LIN {X 0,Y 488.673,Z 877.462,A -85,B 0,C 180,E1 10645.22,E2 10645.22} C_VEL
LIN {X 0,Y 505.067,Z 659.216,A -85,B 0,C 180,E1 10641.829,E2 10641.829} C_VEL
LIN {X 0,Y 508.295,Z 617.041,A -85,B 0,C 180,E1 10641.16,E2 10641.16} C_VEL
LIN {X 0,Y 501.878,Z 605.856,A -85,B 0,C 180,E1 10638.709,E2 10638.709} C_VEL
LIN {X 0,Y 495.396,Z 596.132,A -85,B 0,C 180,E1 10635.872,E2 10635.872} C_VEL
LIN {X 0,Y 491.953,Z 591.127,A -85,B 0,C 180,E1 10634.117,E2 10634.117} C_VEL
LIN {X 0,Y 489.104,Z 586.88,A -85,B 0,C 180,E1 10632.455,E2 10632.455} C_VEL
LIN {X 0,Y 486.126,Z 582.532,A -85,B 0,C 180,E1 10630.428,E2 10630.428} C_VEL
LIN {X 0,Y 483.244,Z 578.317,A -85,B 0,C 180,E1 10627.969,E2 10627.969} C_VEL
LIN {X 0,Y 482.559,Z 577.333,A -85,B 0,C 180,E1 10627.261,E2 10627.261} C_VEL
LIN {X 0,Y 479.956,Z 573.698,A -85,B 0,C 180,E1 10623.464,E2 10623.464} C_VEL
LIN {X 0,Y 479.541,Z 571.93,A -85,B 0,C 180,E1 10621.912,E2 10621.912} C_VEL
LIN {X 0,Y 479.637,Z 572.192,A -85,B 0,C 180,E1 10617.491,E2 10617.491} C_VEL
LIN {X 0,Y 481.251,Z 576.101,A -85,B 0,C 180,E1 10614.037,E2 10614.037} C_VEL
LIN {X 0,Y 483.062,Z 577.924,A -85,B 0,C 180,E1 10612.028,E2 10612.028} C_VEL
LIN {X 0,Y 485.863,Z 582.227,A -85,B 0,C 180,E1 10609.566,E2 10609.566} C_VEL
LIN {X 0,Y 486.983,Z 583.755,A -85,B 0,C 180,E1 10608.752,E2 10608.752} C_VEL
LIN {X 0,Y 490.511,Z 588.903,A -85,B 0,C 180,E1 10606.502,E2 10606.502} C_VEL
LIN {X 0,Y 494.214,Z 594.346,A -85,B 0,C 180,E1 10604.51,E2 10604.51} C_VEL
LIN {X 0,Y 499.508,Z 602.191,A -85,B 0,C 180,E1 10602.075,E2 10602.075} C_VEL
LIN {X 0,Y 505.798,Z 612.068,A -85,B 0,C 180,E1 10599.579,E2 10599.579} C_VEL
LIN {X 0,Y 508.298,Z 616.319,A -85,B 0,C 180,E1 10598.668,E2 10598.668} C_VEL
LIN {X 0,Y 491.94,Z 831.282,A -85,B 0,C 180,E1 10595.331,E2 10595.331} C_VEL
LIN {X 0,Y 486.711,Z 898.786,A -85,B 0,C 180,E1 10594.263,E2 10594.263} C_VEL
LIN {X 0,Y 482.885,Z 928.156,A -85,B 0,C 180,E1 10593.691,E2 10593.691} C_VEL
LIN {X 0,Y 478.634,Z 951.918,A -85,B 0,C 180,E1 10593.081,E2 10593.081} C_VEL
LIN {X 0,Y 474.12,Z 972.963,A -85,B 0,C 180,E1 10592.412,E2 10592.412} C_VEL
LIN {X 0,Y 468.985,Z 993.591,A -85,B 0,C 180,E1 10591.626,E2 10591.626} C_VEL
LIN {X 0,Y 461.912,Z 1018.559,A -85,B 0,C 180,E1 10590.484,E2 10590.484} C_VEL
LIN {X 0,Y 453.841,Z 1042.99,A -85,B 0,C 180,E1 10589.113,E2 10589.113} C_VEL
LIN {X 0,Y 446.612,Z 1062.769,A -85,B 0,C 180,E1 10587.812,E2 10587.812} C_VEL
LIN {X 0,Y 439.339,Z 1081.192,A -85,B 0,C 180,E1 10586.408,E2 10586.408} C_VEL
LIN {X 0,Y 431.297,Z 1100.199,A -85,B 0,C 180,E1 10584.741,E2 10584.741} C_VEL
LIN {X 0,Y 420.775,Z 1123.256,A -85,B 0,C 180,E1 10582.359,E2 10582.359} C_VEL
LIN {X 0,Y 412.35,Z 1140.615,A -85,B 0,C 180,E1 10580.238,E2 10580.238} C_VEL
LIN {X 0,Y 404.56,Z 1156.078,A -85,B 0,C 180,E1 10578.071,E2 10578.071} C_VEL
LIN {X 0,Y 396.87,Z 1170.932,A -85,B 0,C 180,E1 10575.689,E2 10575.689} C_VEL
LIN {X 0,Y 387.854,Z 1188.135,A -85,B 0,C 180,E1 10572.491,E2 10572.491} C_VEL
LIN {X 0,Y 379.872,Z 1203.044,A -85,B 0,C 180,E1 10569.181,E2 10569.181} C_VEL
LIN {X 0,Y 373.901,Z 1214.52,A -85,B 0,C 180,E1 10566.231,E2 10566.231} C_VEL
LIN {X 0,Y 368.717,Z 1224.76,A -85,B 0,C 180,E1 10563.219,E2 10563.219} C_VEL
LIN {X 0,Y 363.893,Z 1234.761,A -85,B 0,C 180,E1 10559.828,E2 10559.828} C_VEL
LIN {X 0,Y 359.105,Z 1245.725,A -85,B 0,C 180,E1 10555.395,E2 10555.395} C_VEL
LIN {X 0,Y 356.135,Z 1253.418,A -85,B 0,C 180,E1 10551.584,E2 10551.584} C_VEL
LIN {X 0,Y 354.269,Z 1259.29,A -85,B 0,C 180,E1 10548.091,E2 10548.091} C_VEL
LIN {X 0,Y 353.032,Z 1264.082,A -85,B 0,C 180,E1 10544.604,E2 10544.604} C_VEL
LIN {X 0,Y 352.351,Z 1267.827,A -85,B 0,C 180,E1 10541.13,E2 10541.13} C_VEL
LIN {X 0,Y 352.013,Z 1270.668,A -85,B 0,C 180,E1 10537.512,E2 10537.512} C_VEL
LIN {X 0,Y 351.926,Z 1272.49,A -85,B 0,C 180,E1 10533.751,E2 10533.751} C_VEL
LIN {X 0,Y 351.896,Z 1273.142,A -85,B 0,C 180,E1 10529.842,E2 10529.842} C_VEL
LIN {X 0,Y 351.929,Z 1272.4,A -85,B 0,C 180,E1 10525.932,E2 10525.932} C_VEL
LIN {X 0,Y 352.019,Z 1270.629,A -85,B 0,C 180,E1 10522.333,E2 10522.333} C_VEL
LIN {X 0,Y 352.334,Z 1267.928,A -85,B 0,C 180,E1 10518.879,E2 10518.879} C_VEL
LIN {X 0,Y 353.012,Z 1264.211,A -85,B 0,C 180,E1 10515.404,E2 10515.404} C_VEL
LIN {X 0,Y 354.153,Z 1259.69,A -85,B 0,C 180,E1 10512.076,E2 10512.076} C_VEL
LIN {X 0,Y 355.968,Z 1253.906,A -85,B 0,C 180,E1 10508.589,E2 10508.589} C_VEL
LIN {X 0,Y 358.586,Z 1246.992,A -85,B 0,C 180,E1 10505.105,E2 10505.105} C_VEL
LIN {X 0,Y 361.326,Z 1240.495,A -85,B 0,C 180,E1 10502.297,E2 10502.297} C_VEL
LIN {X 0,Y 361.626,Z 1237.874,A -85,B 0,C 180,E1 10501.14,E2 10501.14} C_VEL
LIN {X 0,Y 359.431,Z 1230.835,A -85,B 0,C 180,E1 10497.968,E2 10497.968} C_VEL
LIN {X 0,Y 360.102,Z 1228.131,A -85,B 0,C 180,E1 10497.004,E2 10497.004} C_VEL
LIN {X 0,Y 366.407,Z 1216.08,A -85,B 0,C 180,E1 10493.307,E2 10493.307} C_VEL
LIN {X 0,Y 372.543,Z 1204.763,A -85,B 0,C 180,E1 10490.307,E2 10490.307} C_VEL
LIN {X 0,Y 379.15,Z 1192.807,A -85,B 0,C 180,E1 10487.545,E2 10487.545} C_VEL
LIN {X 0,Y 387.197,Z 1178.247,A -85,B 0,C 180,E1 10484.621,E2 10484.621} C_VEL
LIN {X 0,Y 397.614,Z 1158.992,A -85,B 0,C 180,E1 10481.363,E2 10481.363} C_VEL
LIN {X 0,Y 406.081,Z 1142.782,A -85,B 0,C 180,E1 10479.037,E2 10479.037} C_VEL
LIN {X 0,Y 414.037,Z 1126.962,A -85,B 0,C 180,E1 10477.057,E2 10477.057} C_VEL
LIN {X 0,Y 422.44,Z 1109.459,A -85,B 0,C 180,E1 10475.148,E2 10475.148} C_VEL
LIN {X 0,Y 432.786,Z 1086.479,A -85,B 0,C 180,E1 10473.013,E2 10473.013} C_VEL
LIN {X 0,Y 441.432,Z 1065.351,A -85,B 0,C 180,E1 10471.369,E2 10471.369} C_VEL
LIN {X 0,Y 448.646,Z 1046.297,A -85,B 0,C 180,E1 10470.096,E2 10470.096} C_VEL
LIN {X 0,Y 455.36,Z 1026.795,A -85,B 0,C 180,E1 10468.963,E2 10468.963} C_VEL
LIN {X 0,Y 462.1,Z 1005.168,A -85,B 0,C 180,E1 10467.895,E2 10467.895} C_VEL
LIN {X 0,Y 469.494,Z 977.542,A -85,B 0,C 180,E1 10466.775,E2 10466.775} C_VEL
LIN {X 0,Y 474.536,Z 955.094,A -85,B 0,C 180,E1 10466.047,E2 10466.047} C_VEL
LIN {X 0,Y 478.563,Z 933.64,A -85,B 0,C 180,E1 10465.477,E2 10465.477} C_VEL
LIN {X 0,Y 481.975,Z 911.074,A -85,B 0,C 180,E1 10465.003,E2 10465.003} C_VEL
LIN {X 0,Y 485.059,Z 880.548,A -85,B 0,C 180,E1 10464.481,E2 10464.481} C_VEL
LIN {X 0,Y 502.082,Z 660.192,A -85,B 0,C 180,E1 10461.066,E2 10461.066} C_VEL
LIN {X 0,Y 505.159,Z 621.258,A -85,B 0,C 180,E1 10460.454,E2 10460.454} C_VEL
LIN {X 0,Y 498.577,Z 610.88,A -85,B 0,C 180,E1 10457.839,E2 10457.839} C_VEL
LIN {X 0,Y 493.32,Z 602.856,A -85,B 0,C 180,E1 10455.398,E2 10455.398} C_VEL
LIN {X 0,Y 490.433,Z 598.562,A -85,B 0,C 180,E1 10453.861,E2 10453.861} C_VEL
LIN {X 0,Y 487.858,Z 594.642,A -85,B 0,C 180,E1 10452.307,E2 10452.307} C_VEL
LIN {X 0,Y 485.045,Z 590.425,A -85,B 0,C 180,E1 10450.332,E2 10450.332} C_VEL
LIN {X 0,Y 482.19,Z 586.179,A -85,B 0,C 180,E1 10447.806,E2 10447.806} C_VEL
LIN {X 0,Y 481.587,Z 585.291,A -85,B 0,C 180,E1 10447.156,E2 10447.156} C_VEL
LIN {X 0,Y 479.07,Z 581.699,A -85,B 0,C 180,E1 10443.231,E2 10443.231} C_VEL
LIN {X 0,Y 478.717,Z 579.913,A -85,B 0,C 180,E1 10441.556,E2 10441.556} C_VEL
LIN {X 0,Y 478.774,Z 580.143,A -85,B 0,C 180,E1 10438.205,E2 10438.205} C_VEL
LIN {X 0,Y 480.295,Z 584.064,A -85,B 0,C 180,E1 10434.505,E2 10434.505} C_VEL
LIN {X 0,Y 482.075,Z 585.927,A -85,B 0,C 180,E1 10432.432,E2 10432.432} C_VEL
LIN {X 0,Y 484.713,Z 590.12,A -85,B 0,C 180,E1 10430.021,E2 10430.021} C_VEL
LIN {X 0,Y 485.887,Z 591.683,A -85,B 0,C 180,E1 10429.147,E2 10429.147} C_VEL
LIN {X 0,Y 489.137,Z 596.588,A -85,B 0,C 180,E1 10427.005,E2 10427.005} C_VEL
LIN {X 0,Y 492.963,Z 602.326,A -85,B 0,C 180,E1 10424.892,E2 10424.892} C_VEL
LIN {X 0,Y 497.914,Z 609.822,A -85,B 0,C 180,E1 10422.559,E2 10422.559} C_VEL
LIN {X 0,Y 502.016,Z 616.506,A -85,B 0,C 180,E1 10420.844,E2 10420.844} C_VEL
LIN {X 0,Y 505.192,Z 622.48,A -85,B 0,C 180,E1 10419.596,E2 10419.596} C_VEL
LIN {X 0,Y 488.383,Z 838.103,A -85,B 0,C 180,E1 10416.255,E2 10416.255} C_VEL
LIN {X 0,Y 483.187,Z 903.482,A -85,B 0,C 180,E1 10415.22,E2 10415.22} C_VEL
LIN {X 0,Y 479.179,Z 933.314,A -85,B 0,C 180,E1 10414.646,E2 10414.646} C_VEL
LIN {X 0,Y 474.882,Z 956.587,A -85,B 0,C 180,E1 10414.066,E2 10414.066} C_VEL
LIN {X 0,Y 470.159,Z 977.971,A -85,B 0,C 180,E1 10413.403,E2 10413.403} C_VEL
LIN {X 0,Y 464.921,Z 998.45,A -85,B 0,C 180,E1 10412.638,E2 10412.638} C_VEL
LIN {X 0,Y 458.057,Z 1022.054,A -85,B 0,C 180,E1 10411.584,E2 10411.584} C_VEL
LIN {X 0,Y 449.414,Z 1047.74,A -85,B 0,C 180,E1 10410.18,E2 10410.18} C_VEL
LIN {X 0,Y 441.99,Z 1067.639,A -85,B 0,C 180,E1 10408.887,E2 10408.887} C_VEL
LIN {X 0,Y 434.502,Z 1086.202,A -85,B 0,C 180,E1 10407.489,E2 10407.489} C_VEL
LIN {X 0,Y 426.73,Z 1104.125,A -85,B 0,C 180,E1 10405.943,E2 10405.943} C_VEL
LIN {X 0,Y 416.615,Z 1126.069,A -85,B 0,C 180,E1 10403.736,E2 10403.736} C_VEL
LIN {X 0,Y 406.825,Z 1145.735,A -85,B 0,C 180,E1 10401.37,E2 10401.37} C_VEL
LIN {X 0,Y 398.797,Z 1161.288,A -85,B 0,C 180,E1 10399.208,E2 10399.208} C_VEL
LIN {X 0,Y 390.814,Z 1176.347,A -85,B 0,C 180,E1 10396.807,E2 10396.807} C_VEL
LIN {X 0,Y 381.815,Z 1193.118,A -85,B 0,C 180,E1 10393.715,E2 10393.715} C_VEL
LIN {X 0,Y 373.067,Z 1209.073,A -85,B 0,C 180,E1 10390.195,E2 10390.195} C_VEL
LIN {X 0,Y 366.564,Z 1221.218,A -85,B 0,C 180,E1 10387.065,E2 10387.065} C_VEL
LIN {X 0,Y 360.942,Z 1232.107,A -85,B 0,C 180,E1 10383.828,E2 10383.828} C_VEL
LIN {X 0,Y 355.178,Z 1244.038,A -85,B 0,C 180,E1 10379.694,E2 10379.694} C_VEL
LIN {X 0,Y 350.781,Z 1253.927,A -85,B 0,C 180,E1 10375.488,E2 10375.488} C_VEL
LIN {X 0,Y 348.032,Z 1261.068,A -85,B 0,C 180,E1 10371.878,E2 10371.878} C_VEL
LIN {X 0,Y 346.177,Z 1266.915,A -85,B 0,C 180,E1 10368.345,E2 10368.345} C_VEL
LIN {X 0,Y 344.975,Z 1271.541,A -85,B 0,C 180,E1 10364.943,E2 10364.943} C_VEL
LIN {X 0,Y 344.322,Z 1275.199,A -85,B 0,C 180,E1 10361.553,E2 10361.553} C_VEL
LIN {X 0,Y 343.989,Z 1278.028,A -85,B 0,C 180,E1 10358.015,E2 10358.015} C_VEL
LIN {X 0,Y 343.923,Z 1279.699,A -85,B 0,C 180,E1 10354.831,E2 10354.831} C_VEL
LIN {X 0,Y 343.908,Z 1280.543,A -85,B 0,C 180,E1 10351.661,E2 10351.661} C_VEL
LIN {X 0,Y 343.905,Z 1280.564,A -85,B 0,C 180,E1 10348.496,E2 10348.496} C_VEL
LIN {X 0,Y 343.921,Z 1279.761,A -85,B 0,C 180,E1 10345.326,E2 10345.326} C_VEL
LIN {X 0,Y 343.984,Z 1278.131,A -85,B 0,C 180,E1 10342.143,E2 10342.143} C_VEL
LIN {X 0,Y 344.302,Z 1275.345,A -85,B 0,C 180,E1 10338.606,E2 10338.606} C_VEL
LIN {X 0,Y 344.94,Z 1271.729,A -85,B 0,C 180,E1 10335.217,E2 10335.217} C_VEL
LIN {X 0,Y 346.108,Z 1267.147,A -85,B 0,C 180,E1 10331.816,E2 10331.816} C_VEL
LIN {X 0,Y 347.852,Z 1261.567,A -85,B 0,C 180,E1 10328.408,E2 10328.408} C_VEL
LIN {X 0,Y 350.353,Z 1254.956,A -85,B 0,C 180,E1 10325.011,E2 10325.011} C_VEL
LIN {X 0,Y 353.834,Z 1246.86,A -85,B 0,C 180,E1 10321.469,E2 10321.469} C_VEL
LIN {X 0,Y 359.203,Z 1235.669,A -85,B 0,C 180,E1 10317.311,E2 10317.311} C_VEL
LIN {X 0,Y 365.688,Z 1222.885,A -85,B 0,C 180,E1 10313.407,E2 10313.407} C_VEL
LIN {X 0,Y 372.086,Z 1210.809,A -85,B 0,C 180,E1 10310.237,E2 10310.237} C_VEL
LIN {X 0,Y 379.059,Z 1197.97,A -85,B 0,C 180,E1 10307.315,E2 10307.315} C_VEL
LIN {X 0,Y 388.176,Z 1181.321,A -85,B 0,C 180,E1 10304.052,E2 10304.052} C_VEL
LIN {X 0,Y 397.622,Z 1163.448,A -85,B 0,C 180,E1 10301.126,E2 10301.126} C_VEL
LIN {X 0,Y 405.541,Z 1148.136,A -85,B 0,C 180,E1 10298.956,E2 10298.956} C_VEL
LIN {X 0,Y 413.295,Z 1132.58,A -85,B 0,C 180,E1 10297.022,E2 10297.022} C_VEL
LIN {X 0,Y 421.7,Z 1114.95,A -85,B 0,C 180,E1 10295.109,E2 10295.109} C_VEL
LIN {X 0,Y 431.768,Z 1092.578,A -85,B 0,C 180,E1 10293.034,E2 10293.034} C_VEL
LIN {X 0,Y 440.736,Z 1070.608,A -85,B 0,C 180,E1 10291.33,E2 10291.33} C_VEL
LIN {X 0,Y 448.129,Z 1051.038,A -85,B 0,C 180,E1 10290.032,E2 10290.032} C_VEL
LIN {X 0,Y 454.755,Z 1031.833,A -85,B 0,C 180,E1 10288.929,E2 10288.929} C_VEL
LIN {X 0,Y 461.501,Z 1010.238,A -85,B 0,C 180,E1 10287.872,E2 10287.872} C_VEL
LIN {X 0,Y 468.956,Z 982.613,A -85,B 0,C 180,E1 10286.765,E2 10286.765} C_VEL
LIN {X 0,Y 474.149,Z 959.6,A -85,B 0,C 180,E1 10286.027,E2 10286.027} C_VEL
LIN {X 0,Y 478.201,Z 938.258,A -85,B 0,C 180,E1 10285.474,E2 10285.474} C_VEL
LIN {X 0,Y 481.638,Z 915.668,A -85,B 0,C 180,E1 10285.006,E2 10285.006} C_VEL
LIN {X 0,Y 484.693,Z 885.505,A -85,B 0,C 180,E1 10284.489,E2 10284.489} C_VEL
LIN {X 0,Y 501.542,Z 666.545,A -85,B 0,C 180,E1 10281.092,E2 10281.092} C_VEL
LIN {X 0,Y 505.043,Z 622.093,A -85,B 0,C 180,E1 10280.392,E2 10280.392} C_VEL
LIN {X 0,Y 499.654,Z 612.643,A -85,B 0,C 180,E1 10278.251,E2 10278.251} C_VEL
LIN {X 0,Y 493.706,Z 603.514,A -85,B 0,C 180,E1 10275.566,E2 10275.566} C_VEL
LIN {X 0,Y 490.446,Z 598.675,A -85,B 0,C 180,E1 10273.86,E2 10273.86} C_VEL
LIN {X 0,Y 487.658,Z 594.454,A -85,B 0,C 180,E1 10272.192,E2 10272.192} C_VEL
LIN {X 0,Y 484.832,Z 590.256,A -85,B 0,C 180,E1 10270.216,E2 10270.216} C_VEL
LIN {X 0,Y 482.032,Z 586.005,A -85,B 0,C 180,E1 10267.749,E2 10267.749} C_VEL
LIN {X 0,Y 481.027,Z 584.85,A -85,B 0,C 180,E1 10266.685,E2 10266.685} C_VEL
LIN {X 0,Y 478.85,Z 581.273,A -85,B 0,C 180,E1 10263.112,E2 10263.112} C_VEL
LIN {X 0,Y 478.533,Z 579.863,A -85,B 0,C 180,E1 10261.796,E2 10261.796} C_VEL
LIN {X 0,Y 478.629,Z 580.078,A -85,B 0,C 180,E1 10257.605,E2 10257.605} C_VEL
LIN {X 0,Y 480.188,Z 583.98,A -85,B 0,C 180,E1 10254.144,E2 10254.144} C_VEL
LIN {X 0,Y 481.908,Z 585.739,A -85,B 0,C 180,E1 10252.189,E2 10252.189} C_VEL
LIN {X 0,Y 484.732,Z 590.11,A -85,B 0,C 180,E1 10249.662,E2 10249.662} C_VEL
LIN {X 0,Y 486.15,Z 592.291,A -85,B 0,C 180,E1 10248.612,E2 10248.612} C_VEL
LIN {X 0,Y 489.131,Z 596.606,A -85,B 0,C 180,E1 10246.704,E2 10246.704} C_VEL
LIN {X 0,Y 492.773,Z 602.066,A -85,B 0,C 180,E1 10244.705,E2 10244.705} C_VEL
LIN {X 0,Y 497.925,Z 609.877,A -85,B 0,C 180,E1 10242.288,E2 10242.288} C_VEL
LIN {X 0,Y 504.13,Z 619.794,A -85,B 0,C 180,E1 10239.781,E2 10239.781} C_VEL
LIN {X 0,Y 505.034,Z 621.396,A -85,B 0,C 180,E1 10239.439,E2 10239.439} C_VEL
LIN {X 0,Y 488.271,Z 836.362,A -85,B 0,C 180,E1 10236.108,E2 10236.108} C_VEL
LIN {X 0,Y 483.251,Z 899.218,A -85,B 0,C 180,E1 10235.114,E2 10235.114} C_VEL
LIN {X 0,Y 479.184,Z 929.39,A -85,B 0,C 180,E1 10234.525,E2 10234.525} C_VEL
LIN {X 0,Y 474.979,Z 952.343,A -85,B 0,C 180,E1 10233.937,E2 10233.937} C_VEL
LIN {X 0,Y 470.439,Z 973.061,A -85,B 0,C 180,E1 10233.282,E2 10233.282} C_VEL
LIN {X 0,Y 465.241,Z 993.523,A -85,B 0,C 180,E1 10232.509,E2 10232.509} C_VEL
LIN {X 0,Y 458.3,Z 1017.528,A -85,B 0,C 180,E1 10231.422,E2 10231.422} C_VEL
LIN {X 0,Y 450.024,Z 1042.211,A -85,B 0,C 180,E1 10230.06,E2 10230.06} C_VEL
LIN {X 0,Y 442.625,Z 1062.056,A -85,B 0,C 180,E1 10228.766,E2 10228.766} C_VEL
LIN {X 0,Y 435.084,Z 1080.742,A -85,B 0,C 180,E1 10227.352,E2 10227.352} C_VEL
LIN {X 0,Y 427.356,Z 1098.571,A -85,B 0,C 180,E1 10225.804,E2 10225.804} C_VEL
LIN {X 0,Y 417.616,Z 1119.697,A -85,B 0,C 180,E1 10223.678,E2 10223.678} C_VEL
LIN {X 0,Y 407.616,Z 1139.7,A -85,B 0,C 180,E1 10221.269,E2 10221.269} C_VEL
LIN {X 0,Y 399.533,Z 1155.251,A -85,B 0,C 180,E1 10219.098,E2 10219.098} C_VEL
LIN {X 0,Y 391.985,Z 1169.345,A -85,B 0,C 180,E1 10216.851,E2 10216.851} C_VEL
LIN {X 0,Y 384.158,Z 1183.682,A -85,B 0,C 180,E1 10214.234,E2 10214.234} C_VEL
LIN {X 0,Y 375.224,Z 1199.984,A -85,B 0,C 180,E1 10210.762,E2 10210.762} C_VEL
LIN {X 0,Y 367.775,Z 1213.475,A -85,B 0,C 180,E1 10207.325,E2 10207.325} C_VEL
LIN {X 0,Y 361.994,Z 1224.343,A -85,B 0,C 180,E1 10204.109,E2 10204.109} C_VEL
LIN {X 0,Y 357.11,Z 1233.945,A -85,B 0,C 180,E1 10200.827,E2 10200.827} C_VEL
LIN {X 0,Y 352.434,Z 1243.967,A -85,B 0,C 180,E1 10196.818,E2 10196.818} C_VEL
LIN {X 0,Y 348.697,Z 1252.91,A -85,B 0,C 180,E1 10192.423,E2 10192.423} C_VEL
LIN {X 0,Y 346.534,Z 1259.129,A -85,B 0,C 180,E1 10188.684,E2 10188.684} C_VEL
LIN {X 0,Y 345.213,Z 1263.764,A -85,B 0,C 180,E1 10185.287,E2 10185.287} C_VEL
LIN {X 0,Y 344.465,Z 1267.443,A -85,B 0,C 180,E1 10181.898,E2 10181.898} C_VEL
LIN {X 0,Y 344.056,Z 1270.308,A -85,B 0,C 180,E1 10178.36,E2 10178.36} C_VEL
LIN {X 0,Y 343.944,Z 1272.041,A -85,B 0,C 180,E1 10175.175,E2 10175.175} C_VEL
LIN {X 0,Y 343.913,Z 1272.968,A -85,B 0,C 180,E1 10172.004,E2 10172.004} C_VEL
LIN {X 0,Y 343.888,Z 1273.095,A -85,B 0,C 180,E1 10168.839,E2 10168.839} C_VEL
LIN {X 0,Y 343.932,Z 1272.353,A -85,B 0,C 180,E1 10165.503,E2 10165.503} C_VEL
LIN {X 0,Y 344.023,Z 1270.717,A -85,B 0,C 180,E1 10162.154,E2 10162.154} C_VEL
LIN {X 0,Y 344.373,Z 1268.017,A -85,B 0,C 180,E1 10158.618,E2 10158.618} C_VEL
LIN {X 0,Y 345.058,Z 1264.504,A -85,B 0,C 180,E1 10155.232,E2 10155.232} C_VEL
LIN {X 0,Y 346.269,Z 1260.005,A -85,B 0,C 180,E1 10151.81,E2 10151.81} C_VEL
LIN {X 0,Y 348.165,Z 1254.296,A -85,B 0,C 180,E1 10148.261,E2 10148.261} C_VEL
LIN {X 0,Y 350.757,Z 1247.782,A -85,B 0,C 180,E1 10144.872,E2 10144.872} C_VEL
LIN {X 0,Y 354.526,Z 1239.394,A -85,B 0,C 180,E1 10141.172,E2 10141.172} C_VEL
LIN {X 0,Y 360.102,Z 1228.131,A -85,B 0,C 180,E1 10137.004,E2 10137.004} C_VEL
LIN {X 0,Y 360.852,Z 1224.964,A -85,B 0,C 180,E1 10135.886,E2 10135.886} C_VEL
LIN {X 0,Y 359.897,Z 1217.295,A -85,B 0,C 180,E1 10132.928,E2 10132.928} C_VEL
LIN {X 0,Y 361.031,Z 1213.805,A -85,B 0,C 180,E1 10131.835,E2 10131.835} C_VEL
LIN {X 0,Y 369.435,Z 1199.299,A -85,B 0,C 180,E1 10128.099,E2 10128.099} C_VEL
LIN {X 0,Y 378.439,Z 1183.444,A -85,B 0,C 180,E1 10124.714,E2 10124.714} C_VEL
LIN {X 0,Y 386.113,Z 1169.91,A -85,B 0,C 180,E1 10122.224,E2 10122.224} C_VEL
LIN {X 0,Y 393.936,Z 1155.806,A -85,B 0,C 180,E1 10119.954,E2 10119.954} C_VEL
LIN {X 0,Y 402.042,Z 1140.729,A -85,B 0,C 180,E1 10117.831,E2 10117.831} C_VEL
LIN {X 0,Y 411.334,Z 1122.726,A -85,B 0,C 180,E1 10115.631,E2 10115.631} C_VEL
LIN {X 0,Y 422.245,Z 1100.052,A -85,B 0,C 180,E1 10113.3,E2 10113.3} C_VEL
LIN {X 0,Y 430.24,Z 1082.169,A -85,B 0,C 180,E1 10111.736,E2 10111.736} C_VEL
LIN {X 0,Y 437.872,Z 1063.817,A -85,B 0,C 180,E1 10110.338,E2 10110.338} C_VEL
LIN {X 0,Y 445.433,Z 1044.138,A -85,B 0,C 180,E1 10109.047,E2 10109.047} C_VEL
LIN {X 0,Y 453.195,Z 1021.864,A -85,B 0,C 180,E1 10107.795,E2 10107.795} C_VEL
LIN {X 0,Y 461.151,Z 995.561,A -85,B 0,C 180,E1 10106.582,E2 10106.582} C_VEL
LIN {X 0,Y 466.66,Z 974.518,A -85,B 0,C 180,E1 10105.783,E2 10105.783} C_VEL
LIN {X 0,Y 471.412,Z 953.438,A -85,B 0,C 180,E1 10105.116,E2 10105.116} C_VEL
LIN {X 0,Y 475.529,Z 931.632,A -85,B 0,C 180,E1 10104.554,E2 10104.554} C_VEL
LIN {X 0,Y 479.571,Z 904.31,A -85,B 0,C 180,E1 10104.003,E2 10104.003} C_VEL
LIN {X 0,Y 483.419,Z 859.466,A -85,B 0,C 180,E1 10103.284,E2 10103.284} C_VEL
LIN {X 0,Y 500.832,Z 640.859,A -85,B 0,C 180,E1 10099.906,E2 10099.906} C_VEL
LIN {X 0,Y 501.967,Z 626.544,A -85,B 0,C 180,E1 10099.672,E2 10099.672} C_VEL
LIN {X 0,Y 495.879,Z 616.663,A -85,B 0,C 180,E1 10097.121,E2 10097.121} C_VEL
LIN {X 0,Y 489.971,Z 607.504,A -85,B 0,C 180,E1 10094.175,E2 10094.175} C_VEL
LIN {X 0,Y 486.334,Z 602.099,A -85,B 0,C 180,E1 10091.985,E2 10091.985} C_VEL
LIN {X 0,Y 483.758,Z 598.151,A -85,B 0,C 180,E1 10090.119,E2 10090.119} C_VEL
LIN {X 0,Y 480.989,Z 593.868,A -85,B 0,C 180,E1 10087.586,E2 10087.586} C_VEL
LIN {X 0,Y 479.876,Z 592.633,A -85,B 0,C 180,E1 10086.34,E2 10086.34} C_VEL
LIN {X 0,Y 477.92,Z 589.022,A -85,B 0,C 180,E1 10082.638,E2 10082.638} C_VEL
LIN {X 0,Y 477.718,Z 587.847,A -85,B 0,C 180,E1 10081.439,E2 10081.439} C_VEL
LIN {X 0,Y 477.776,Z 588.022,A -85,B 0,C 180,E1 10078.321,E2 10078.321} C_VEL
LIN {X 0,Y 479.319,Z 592.044,A -85,B 0,C 180,E1 10074.493,E2 10074.493} C_VEL
LIN {X 0,Y 480.927,Z 593.741,A -85,B 0,C 180,E1 10072.594,E2 10072.594} C_VEL
LIN {X 0,Y 483.586,Z 598.002,A -85,B 0,C 180,E1 10070.118,E2 10070.118} C_VEL
LIN {X 0,Y 484.814,Z 599.794,A -85,B 0,C 180,E1 10069.183,E2 10069.183} C_VEL
LIN {X 0,Y 487.86,Z 604.449,A -85,B 0,C 180,E1 10067.151,E2 10067.151} C_VEL
LIN {X 0,Y 491.42,Z 609.869,A -85,B 0,C 180,E1 10065.145,E2 10065.145} C_VEL
LIN {X 0,Y 496.404,Z 617.608,A -85,B 0,C 180,E1 10062.746,E2 10062.746} C_VEL
LIN {X 0,Y 500.246,Z 624.005,A -85,B 0,C 180,E1 10061.107,E2 10061.107} C_VEL
LIN {X 0,Y 502.019,Z 627.563,A -85,B 0,C 180,E1 10060.377,E2 10060.377} C_VEL
LIN {X 0,Y 484.82,Z 842.961,A -85,B 0,C 180,E1 10057.048,E2 10057.048} C_VEL
LIN {X 0,Y 479.833,Z 903.843,A -85,B 0,C 180,E1 10056.084,E2 10056.084} C_VEL
LIN {X 0,Y 475.608,Z 934.264,A -85,B 0,C 180,E1 10055.498,E2 10055.498} C_VEL
LIN {X 0,Y 471.345,Z 956.834,A -85,B 0,C 180,E1 10054.937,E2 10054.937} C_VEL
LIN {X 0,Y 466.595,Z 977.892,A -85,B 0,C 180,E1 10054.29,E2 10054.29} C_VEL
LIN {X 0,Y 461.251,Z 998.369,A -85,B 0,C 180,E1 10053.532,E2 10053.532} C_VEL
LIN {X 0,Y 454.266,Z 1021.883,A -85,B 0,C 180,E1 10052.491,E2 10052.491} C_VEL
LIN {X 0,Y 445.773,Z 1046.663,A -85,B 0,C 180,E1 10051.153,E2 10051.153} C_VEL
LIN {X 0,Y 438.136,Z 1066.741,A -85,B 0,C 180,E1 10049.863,E2 10049.863} C_VEL
LIN {X 0,Y 430.588,Z 1085.045,A -85,B 0,C 180,E1 10048.501,E2 10048.501} C_VEL
LIN {X 0,Y 422.675,Z 1102.864,A -85,B 0,C 180,E1 10046.983,E2 10046.983} C_VEL
LIN {X 0,Y 413.256,Z 1122.823,A -85,B 0,C 180,E1 10045.01,E2 10045.01} C_VEL
LIN {X 0,Y 402.261,Z 1144.517,A -85,B 0,C 180,E1 10042.45,E2 10042.45} C_VEL
LIN {X 0,Y 393.587,Z 1160.794,A -85,B 0,C 180,E1 10040.193,E2 10040.193} C_VEL
LIN {X 0,Y 385.234,Z 1176.026,A -85,B 0,C 180,E1 10037.759,E2 10037.759} C_VEL
LIN {X 0,Y 376.223,Z 1192.201,A -85,B 0,C 180,E1 10034.763,E2 10034.763} C_VEL
LIN {X 0,Y 367.121,Z 1208.242,A -85,B 0,C 180,E1 10031.224,E2 10031.224} C_VEL
LIN {X 0,Y 360.199,Z 1220.55,A -85,B 0,C 180,E1 10028.035,E2 10028.035} C_VEL
LIN {X 0,Y 354.294,Z 1231.393,A -85,B 0,C 180,E1 10024.788,E2 10024.788} C_VEL
LIN {X 0,Y 349.017,Z 1241.642,A -85,B 0,C 180,E1 10021.227,E2 10021.227} C_VEL
LIN {X 0,Y 343.59,Z 1253.123,A -85,B 0,C 180,E1 10016.433,E2 10016.433} C_VEL
LIN {X 0,Y 340.506,Z 1260.591,A -85,B 0,C 180,E1 10012.617,E2 10012.617} C_VEL
LIN {X 0,Y 338.431,Z 1266.568,A -85,B 0,C 180,E1 10008.959,E2 10008.959} C_VEL
LIN {X 0,Y 337.096,Z 1271.314,A -85,B 0,C 180,E1 10005.417,E2 10005.417} C_VEL
LIN {X 0,Y 336.385,Z 1274.949,A -85,B 0,C 180,E1 10002.004,E2 10002.004} C_VEL
LIN {X 0,Y 336.029,Z 1277.71,A -85,B 0,C 180,E1 9998.551,E2 9998.551} C_VEL
LIN {X 0,Y 335.929,Z 1279.474,A -85,B 0,C 180,E1 9995.289,E2 9995.289} C_VEL
LIN {X 0,Y 335.912,Z 1280.41,A -85,B 0,C 180,E1 9992.042,E2 9992.042} C_VEL
LIN {X 0,Y 335.892,Z 1280.522,A -85,B 0,C 180,E1 9988.801,E2 9988.801} C_VEL
LIN {X 0,Y 335.921,Z 1279.742,A -85,B 0,C 180,E1 9985.386,E2 9985.386} C_VEL
LIN {X 0,Y 335.991,Z 1278.043,A -85,B 0,C 180,E1 9981.955,E2 9981.955} C_VEL
LIN {X 0,Y 336.336,Z 1275.255,A -85,B 0,C 180,E1 9978.332,E2 9978.332} C_VEL
LIN {X 0,Y 337.022,Z 1271.639,A -85,B 0,C 180,E1 9974.861,E2 9974.861} C_VEL
LIN {X 0,Y 338.284,Z 1267.056,A -85,B 0,C 180,E1 9971.38,E2 9971.38} C_VEL
LIN {X 0,Y 340.227,Z 1261.28,A -85,B 0,C 180,E1 9967.783,E2 9967.783} C_VEL
LIN {X 0,Y 342.959,Z 1254.507,A -85,B 0,C 180,E1 9964.249,E2 9964.249} C_VEL
LIN {X 0,Y 346.89,Z 1245.95,A -85,B 0,C 180,E1 9960.465,E2 9960.465} C_VEL
LIN {X 0,Y 353.46,Z 1232.996,A -85,B 0,C 180,E1 9955.737,E2 9955.737} C_VEL
LIN {X 0,Y 359.261,Z 1222.214,A -85,B 0,C 180,E1 9952.442,E2 9952.442} C_VEL
LIN {X 0,Y 365.654,Z 1210.715,A -85,B 0,C 180,E1 9949.393,E2 9949.393} C_VEL
LIN {X 0,Y 373.202,Z 1197.393,A -85,B 0,C 180,E1 9946.335,E2 9946.335} C_VEL
LIN {X 0,Y 382.99,Z 1180.102,A -85,B 0,C 180,E1 9942.954,E2 9942.954} C_VEL
LIN {X 0,Y 392.392,Z 1162.918,A -85,B 0,C 180,E1 9940.138,E2 9940.138} C_VEL
LIN {X 0,Y 400.672,Z 1147.412,A -85,B 0,C 180,E1 9937.943,E2 9937.943} C_VEL
LIN {X 0,Y 408.909,Z 1131.371,A -85,B 0,C 180,E1 9935.961,E2 9935.961} C_VEL
LIN {X 0,Y 418.494,Z 1111.803,A -85,B 0,C 180,E1 9933.871,E2 9933.871} C_VEL
LIN {X 0,Y 428.576,Z 1089.536,A -85,B 0,C 180,E1 9931.869,E2 9931.869} C_VEL
LIN {X 0,Y 436.847,Z 1069.701,A -85,B 0,C 180,E1 9930.353,E2 9930.353} C_VEL
LIN {X 0,Y 444.418,Z 1050.041,A -85,B 0,C 180,E1 9929.061,E2 9929.061} C_VEL
LIN {X 0,Y 451.525,Z 1029.814,A -85,B 0,C 180,E1 9927.921,E2 9927.921} C_VEL
LIN {X 0,Y 459.519,Z 1004.322,A -85,B 0,C 180,E1 9926.716,E2 9926.716} C_VEL
LIN {X 0,Y 466.078,Z 979.553,A -85,B 0,C 180,E1 9925.774,E2 9925.774} C_VEL
LIN {X 0,Y 471.018,Z 957.822,A -85,B 0,C 180,E1 9925.097,E2 9925.097} C_VEL
LIN {X 0,Y 475.143,Z 936.199,A -85,B 0,C 180,E1 9924.553,E2 9924.553} C_VEL
LIN {X 0,Y 479.216,Z 908.868,A -85,B 0,C 180,E1 9924.006,E2 9924.006} C_VEL
LIN {X 0,Y 483.031,Z 864.362,A -85,B 0,C 180,E1 9923.291,E2 9923.291} C_VEL
LIN {X 0,Y 500.234,Z 647.553,A -85,B 0,C 180,E1 9919.937,E2 9919.937} C_VEL
LIN {X 0,Y 501.874,Z 627.214,A -85,B 0,C 180,E1 9919.615,E2 9919.615} C_VEL
LIN {X 0,Y 497.726,Z 619.81,A -85,B 0,C 180,E1 9917.901,E2 9917.901} C_VEL
LIN {X 0,Y 491.917,Z 610.731,A -85,B 0,C 180,E1 9915.201,E2 9915.201} C_VEL
LIN {X 0,Y 488.847,Z 606.077,A -85,B 0,C 180,E1 9913.544,E2 9913.544} C_VEL
LIN {X 0,Y 486.222,Z 602.027,A -85,B 0,C 180,E1 9911.928,E2 9911.928} C_VEL
LIN {X 0,Y 483.544,Z 597.977,A -85,B 0,C 180,E1 9910.003,E2 9910.003} C_VEL
LIN {X 0,Y 480.776,Z 593.568,A -85,B 0,C 180,E1 9907.469,E2 9907.469} C_VEL
LIN {X 0,Y 477.865,Z 589.307,A -85,B 0,C 180,E1 9903.119,E2 9903.119} C_VEL
LIN {X 0,Y 477.528,Z 587.796,A -85,B 0,C 180,E1 9901.68,E2 9901.68} C_VEL
LIN {X 0,Y 477.622,Z 587.965,A -85,B 0,C 180,E1 9897.72,E2 9897.72} C_VEL
LIN {X 0,Y 479.212,Z 591.967,A -85,B 0,C 180,E1 9894.132,E2 9894.132} C_VEL
LIN {X 0,Y 480.809,Z 593.677,A -85,B 0,C 180,E1 9892.291,E2 9892.291} C_VEL
LIN {X 0,Y 483.761,Z 598.153,A -85,B 0,C 180,E1 9889.641,E2 9889.641} C_VEL
LIN {X 0,Y 487.757,Z 604.309,A -85,B 0,C 180,E1 9886.908,E2 9886.908} C_VEL
LIN {X 0,Y 491.338,Z 609.783,A -85,B 0,C 180,E1 9884.901,E2 9884.901} C_VEL
LIN {X 0,Y 496.475,Z 617.768,A -85,B 0,C 180,E1 9882.447,E2 9882.447} C_VEL
LIN {X 0,Y 501.855,Z 626.561,A -85,B 0,C 180,E1 9880.219,E2 9880.219} C_VEL
LIN {X 0,Y 484.687,Z 841.484,A -85,B 0,C 180,E1 9876.898,E2 9876.898} C_VEL
LIN {X 0,Y 479.879,Z 899.863,A -85,B 0,C 180,E1 9875.974,E2 9875.974} C_VEL
LIN {X 0,Y 475.699,Z 929.987,A -85,B 0,C 180,E1 9875.386,E2 9875.386} C_VEL
LIN {X 0,Y 471.453,Z 952.658,A -85,B 0,C 180,E1 9874.81,E2 9874.81} C_VEL
LIN {X 0,Y 466.869,Z 973.159,A -85,B 0,C 180,E1 9874.166,E2 9874.166} C_VEL
LIN {X 0,Y 461.744,Z 992.964,A -85,B 0,C 180,E1 9873.426,E2 9873.426} C_VEL
LIN {X 0,Y 455.495,Z 1014.241,A -85,B 0,C 180,E1 9872.482,E2 9872.482} C_VEL
LIN {X 0,Y 446.679,Z 1040.512,A -85,B 0,C 180,E1 9871.077,E2 9871.077} C_VEL
LIN {X 0,Y 438.442,Z 1062.151,A -85,B 0,C 180,E1 9869.679,E2 9869.679} C_VEL
LIN {X 0,Y 430.797,Z 1080.649,A -85,B 0,C 180,E1 9868.286,E2 9868.286} C_VEL
LIN {X 0,Y 423.082,Z 1098.001,A -85,B 0,C 180,E1 9866.788,E2 9866.788} C_VEL
LIN {X 0,Y 413.906,Z 1117.37,A -85,B 0,C 180,E1 9864.861,E2 9864.861} C_VEL
LIN {X 0,Y 403.009,Z 1138.786,A -85,B 0,C 180,E1 9862.325,E2 9862.325} C_VEL
LIN {X 0,Y 394.476,Z 1154.701,A -85,B 0,C 180,E1 9860.112,E2 9860.112} C_VEL
LIN {X 0,Y 386.316,Z 1169.44,A -85,B 0,C 180,E1 9857.756,E2 9857.756} C_VEL
LIN {X 0,Y 378.104,Z 1183.96,A -85,B 0,C 180,E1 9855.083,E2 9855.083} C_VEL
LIN {X 0,Y 368.541,Z 1200.708,A -85,B 0,C 180,E1 9851.456,E2 9851.456} C_VEL
LIN {X 0,Y 360.818,Z 1214.138,A -85,B 0,C 180,E1 9847.97,E2 9847.97} C_VEL
LIN {X 0,Y 355.077,Z 1224.437,A -85,B 0,C 180,E1 9844.869,E2 9844.869} C_VEL
LIN {X 0,Y 349.964,Z 1234.038,A -85,B 0,C 180,E1 9841.528,E2 9841.528} C_VEL
LIN {X 0,Y 344.847,Z 1244.461,A -85,B 0,C 180,E1 9837.27,E2 9837.27} C_VEL
LIN {X 0,Y 340.933,Z 1253.301,A -85,B 0,C 180,E1 9832.78,E2 9832.78} C_VEL
LIN {X 0,Y 338.738,Z 1259.22,A -85,B 0,C 180,E1 9829.13,E2 9829.13} C_VEL
LIN {X 0,Y 337.328,Z 1263.854,A -85,B 0,C 180,E1 9825.653,E2 9825.653} C_VEL
LIN {X 0,Y 336.512,Z 1267.557,A -85,B 0,C 180,E1 9822.157,E2 9822.157} C_VEL
LIN {X 0,Y 336.077,Z 1270.397,A -85,B 0,C 180,E1 9818.56,E2 9818.56} C_VEL
LIN {X 0,Y 335.948,Z 1272.129,A -85,B 0,C 180,E1 9815.299,E2 9815.299} C_VEL
LIN {X 0,Y 335.913,Z 1273.056,A -85,B 0,C 180,E1 9812.052,E2 9812.052} C_VEL
LIN {X 0,Y 335.89,Z 1273.182,A -85,B 0,C 180,E1 9808.811,E2 9808.811} C_VEL
LIN {X 0,Y 335.933,Z 1272.44,A -85,B 0,C 180,E1 9805.396,E2 9805.396} C_VEL
LIN {X 0,Y 336.034,Z 1270.804,A -85,B 0,C 180,E1 9801.966,E2 9801.966} C_VEL
LIN {X 0,Y 336.413,Z 1268.105,A -85,B 0,C 180,E1 9798.345,E2 9798.345} C_VEL
LIN {X 0,Y 337.149,Z 1264.592,A -85,B 0,C 180,E1 9794.877,E2 9794.877} C_VEL
LIN {X 0,Y 338.454,Z 1260.129,A -85,B 0,C 180,E1 9791.4,E2 9791.4} C_VEL
LIN {X 0,Y 340.491,Z 1254.385,A -85,B 0,C 180,E1 9787.746,E2 9787.746} C_VEL
LIN {X 0,Y 343.239,Z 1247.871,A -85,B 0,C 180,E1 9784.282,E2 9784.282} C_VEL
LIN {X 0,Y 347.23,Z 1239.484,A -85,B 0,C 180,E1 9780.508,E2 9780.508} C_VEL
LIN {X 0,Y 353.626,Z 1227.232,A -85,B 0,C 180,E1 9775.942,E2 9775.942} C_VEL
LIN {X 0,Y 360.017,Z 1215.601,A -85,B 0,C 180,E1 9772.345,E2 9772.345} C_VEL
LIN {X 0,Y 361.031,Z 1213.805,A -85,B 0,C 180,E1 9771.835,E2 9771.835} C_VEL
LIN {X 0,Y 362.283,Z 1210.341,A -85,B 0,C 180,E1 9770.755,E2 9770.755} C_VEL
LIN {X 0,Y 362.775,Z 1201.18,A -85,B 0,C 180,E1 9767.724,E2 9767.724} C_VEL
LIN {X 0,Y 364.154,Z 1197.772,A -85,B 0,C 180,E1 9766.848,E2 9766.848} C_VEL
LIN {X 0,Y 372.593,Z 1183.533,A -85,B 0,C 180,E1 9763.799,E2 9763.799} C_VEL
LIN {X 0,Y 380.703,Z 1169.715,A -85,B 0,C 180,E1 9761.242,E2 9761.242} C_VEL
LIN {X 0,Y 389.452,Z 1154.433,A -85,B 0,C 180,E1 9758.789,E2 9758.789} C_VEL
LIN {X 0,Y 400.004,Z 1135.389,A -85,B 0,C 180,E1 9756.168,E2 9756.168} C_VEL
LIN {X 0,Y 410.742,Z 1114.479,A -85,B 0,C 180,E1 9753.776,E2 9753.776} C_VEL
LIN {X 0,Y 419.319,Z 1096.811,A -85,B 0,C 180,E1 9752.049,E2 9752.049} C_VEL
LIN {X 0,Y 427.273,Z 1079.324,A -85,B 0,C 180,E1 9750.563,E2 9750.563} C_VEL
LIN {X 0,Y 435.43,Z 1059.955,A -85,B 0,C 180,E1 9749.132,E2 9749.132} C_VEL
LIN {X 0,Y 445.3,Z 1033.978,A -85,B 0,C 180,E1 9747.522,E2 9747.522} C_VEL
LIN {X 0,Y 452.614,Z 1012.098,A -85,B 0,C 180,E1 9746.401,E2 9746.401} C_VEL
LIN {X 0,Y 458.661,Z 991.794,A -85,B 0,C 180,E1 9745.522,E2 9745.522} C_VEL
LIN {X 0,Y 464.079,Z 971.05,A -85,B 0,C 180,E1 9744.764,E2 9744.764} C_VEL
LIN {X 0,Y 469.583,Z 946.366,A -85,B 0,C 180,E1 9744.025,E2 9744.025} C_VEL
LIN {X 0,Y 474.379,Z 918.514,A -85,B 0,C 180,E1 9743.388,E2 9743.388} C_VEL
LIN {X 0,Y 477.244,Z 895.559,A -85,B 0,C 180,E1 9742.975,E2 9742.975} C_VEL
LIN {X 0,Y 494.479,Z 684.942,A -85,B 0,C 180,E1 9739.713,E2 9739.713} C_VEL
LIN {X 0,Y 498.887,Z 631.81,A -85,B 0,C 180,E1 9738.886,E2 9738.886} C_VEL
LIN {X 0,Y 493.168,Z 622.616,A -85,B 0,C 180,E1 9736.369,E2 9736.369} C_VEL
LIN {X 0,Y 488.467,Z 615.059,A -85,B 0,C 180,E1 9733.917,E2 9733.917} C_VEL
LIN {X 0,Y 484.914,Z 609.671,A -85,B 0,C 180,E1 9731.719,E2 9731.719} C_VEL
LIN {X 0,Y 482.478,Z 605.874,A -85,B 0,C 180,E1 9729.905,E2 9729.905} C_VEL
LIN {X 0,Y 479.746,Z 601.434,A -85,B 0,C 180,E1 9727.304,E2 9727.304} C_VEL
LIN {X 0,Y 476.998,Z 597.311,A -85,B 0,C 180,E1 9722.884,E2 9722.884} C_VEL
LIN {X 0,Y 476.721,Z 595.782,A -85,B 0,C 180,E1 9721.322,E2 9721.322} C_VEL
LIN {X 0,Y 476.791,Z 596.046,A -85,B 0,C 180,E1 9718.318,E2 9718.318} C_VEL
LIN {X 0,Y 478.344,Z 600.027,A -85,B 0,C 180,E1 9714.482,E2 9714.482} C_VEL
LIN {X 0,Y 479.832,Z 601.676,A -85,B 0,C 180,E1 9712.697,E2 9712.697} C_VEL
LIN {X 0,Y 482.613,Z 606.042,A -85,B 0,C 180,E1 9710.098,E2 9710.098} C_VEL
LIN {X 0,Y 486.314,Z 611.833,A -85,B 0,C 180,E1 9707.472,E2 9707.472} C_VEL
LIN {X 0,Y 489.993,Z 617.583,A -85,B 0,C 180,E1 9705.343,E2 9705.343} C_VEL
LIN {X 0,Y 494.899,Z 625.388,A -85,B 0,C 180,E1 9702.935,E2 9702.935} C_VEL
LIN {X 0,Y 498.488,Z 631.501,A -85,B 0,C 180,E1 9701.371,E2 9701.371} C_VEL
LIN {X 0,Y 498.942,Z 632.637,A -85,B 0,C 180,E1 9701.168,E2 9701.168} C_VEL
LIN {X 0,Y 481.294,Z 848.543,A -85,B 0,C 180,E1 9697.84,E2 9697.84} C_VEL
LIN {X 0,Y 476.567,Z 904.418,A -85,B 0,C 180,E1 9696.957,E2 9696.957} C_VEL
LIN {X 0,Y 472.305,Z 934.319,A -85,B 0,C 180,E1 9696.383,E2 9696.383} C_VEL
LIN {X 0,Y 467.965,Z 956.865,A -85,B 0,C 180,E1 9695.828,E2 9695.828} C_VEL
LIN {X 0,Y 463.147,Z 977.812,A -85,B 0,C 180,E1 9695.191,E2 9695.191} C_VEL
LIN {X 0,Y 457.696,Z 998.288,A -85,B 0,C 180,E1 9694.441,E2 9694.441} C_VEL
LIN {X 0,Y 450.566,Z 1021.8,A -85,B 0,C 180,E1 9693.409,E2 9693.409} C_VEL
LIN {X 0,Y 441.749,Z 1046.94,A -85,B 0,C 180,E1 9692.06,E2 9692.06} C_VEL
LIN {X 0,Y 433.756,Z 1067.437,A -85,B 0,C 180,E1 9690.745,E2 9690.745} C_VEL
LIN {X 0,Y 426.193,Z 1085.293,A -85,B 0,C 180,E1 9689.419,E2 9689.419} C_VEL
LIN {X 0,Y 417.913,Z 1103.447,A -85,B 0,C 180,E1 9687.872,E2 9687.872} C_VEL
LIN {X 0,Y 407.585,Z 1124.743,A -85,B 0,C 180,E1 9685.753,E2 9685.753} C_VEL
LIN {X 0,Y 397.004,Z 1144.837,A -85,B 0,C 180,E1 9683.351,E2 9683.351} C_VEL
LIN {X 0,Y 388.051,Z 1161.11,A -85,B 0,C 180,E1 9681.082,E2 9681.082} C_VEL
LIN {X 0,Y 379.505,Z 1176.168,A -85,B 0,C 180,E1 9678.658,E2 9678.658} C_VEL
LIN {X 0,Y 369.864,Z 1192.885,A -85,B 0,C 180,E1 9675.527,E2 9675.527} C_VEL
LIN {X 0,Y 360.45,Z 1208.79,A -85,B 0,C 180,E1 9671.945,E2 9671.945} C_VEL
LIN {X 0,Y 353.272,Z 1221.037,A -85,B 0,C 180,E1 9668.711,E2 9668.711} C_VEL
LIN {X 0,Y 347.069,Z 1231.925,A -85,B 0,C 180,E1 9665.377,E2 9665.377} C_VEL
LIN {X 0,Y 340.938,Z 1243.402,A -85,B 0,C 180,E1 9661.264,E2 9661.264} C_VEL
LIN {X 0,Y 335.778,Z 1253.769,A -85,B 0,C 180,E1 9656.702,E2 9656.702} C_VEL
LIN {X 0,Y 332.735,Z 1260.808,A -85,B 0,C 180,E1 9652.989,E2 9652.989} C_VEL
LIN {X 0,Y 330.547,Z 1266.736,A -85,B 0,C 180,E1 9649.246,E2 9649.246} C_VEL
LIN {X 0,Y 329.157,Z 1271.406,A -85,B 0,C 180,E1 9645.642,E2 9645.642} C_VEL
LIN {X 0,Y 328.402,Z 1275.022,A -85,B 0,C 180,E1 9642.122,E2 9642.122} C_VEL
LIN {X 0,Y 328.031,Z 1277.737,A -85,B 0,C 180,E1 9638.584,E2 9638.584} C_VEL
LIN {X 0,Y 327.928,Z 1279.455,A -85,B 0,C 180,E1 9635.243,E2 9635.243} C_VEL
LIN {X 0,Y 327.911,Z 1280.345,A -85,B 0,C 180,E1 9631.917,E2 9631.917} C_VEL
LIN {X 0,Y 327.901,Z 1280.412,A -85,B 0,C 180,E1 9628.597,E2 9628.597} C_VEL
LIN {X 0,Y 327.922,Z 1279.654,A -85,B 0,C 180,E1 9625.273,E2 9625.273} C_VEL
LIN {X 0,Y 328.003,Z 1277.954,A -85,B 0,C 180,E1 9621.758,E2 9621.758} C_VEL
LIN {X 0,Y 328.375,Z 1275.166,A -85,B 0,C 180,E1 9618.046,E2 9618.046} C_VEL
LIN {X 0,Y 329.119,Z 1271.549,A -85,B 0,C 180,E1 9614.489,E2 9614.489} C_VEL
LIN {X 0,Y 330.472,Z 1266.965,A -85,B 0,C 180,E1 9610.923,E2 9610.923} C_VEL
LIN {X 0,Y 332.485,Z 1261.384,A -85,B 0,C 180,E1 9607.356,E2 9607.356} C_VEL
LIN {X 0,Y 335.298,Z 1254.771,A -85,B 0,C 180,E1 9603.806,E2 9603.806} C_VEL
LIN {X 0,Y 339.196,Z 1246.674,A -85,B 0,C 180,E1 9600.116,E2 9600.116} C_VEL
LIN {X 0,Y 345.184,Z 1235.483,A -85,B 0,C 180,E1 9595.805,E2 9595.805} C_VEL
LIN {X 0,Y 352.293,Z 1222.697,A -85,B 0,C 180,E1 9591.772,E2 9591.772} C_VEL
LIN {X 0,Y 359.312,Z 1210.621,A -85,B 0,C 180,E1 9588.52,E2 9588.52} C_VEL
LIN {X 0,Y 366.873,Z 1197.782,A -85,B 0,C 180,E1 9585.534,E2 9585.534} C_VEL
LIN {X 0,Y 376.862,Z 1180.836,A -85,B 0,C 180,E1 9582.165,E2 9582.165} C_VEL
LIN {X 0,Y 386.538,Z 1163.739,A -85,B 0,C 180,E1 9579.328,E2 9579.328} C_VEL
LIN {X 0,Y 395.316,Z 1147.827,A -85,B 0,C 180,E1 9577.057,E2 9577.057} C_VEL
LIN {X 0,Y 403.5,Z 1132.391,A -85,B 0,C 180,E1 9575.136,E2 9575.136} C_VEL
LIN {X 0,Y 412.089,Z 1115.372,A -85,B 0,C 180,E1 9573.288,E2 9573.288} C_VEL
LIN {X 0,Y 422.366,Z 1093.824,A -85,B 0,C 180,E1 9571.28,E2 9571.28} C_VEL
LIN {X 0,Y 432.093,Z 1071.233,A -85,B 0,C 180,E1 9569.528,E2 9569.528} C_VEL
LIN {X 0,Y 440.036,Z 1051.178,A -85,B 0,C 180,E1 9568.206,E2 9568.206} C_VEL
LIN {X 0,Y 447.065,Z 1031.733,A -85,B 0,C 180,E1 9567.105,E2 9567.105} C_VEL
LIN {X 0,Y 453.881,Z 1010.836,A -85,B 0,C 180,E1 9566.095,E2 9566.095} C_VEL
LIN {X 0,Y 461.534,Z 983.9,A -85,B 0,C 180,E1 9565.023,E2 9565.023} C_VEL
LIN {X 0,Y 467.194,Z 959.884,A -85,B 0,C 180,E1 9564.263,E2 9564.263} C_VEL
LIN {X 0,Y 471.434,Z 938.448,A -85,B 0,C 180,E1 9563.718,E2 9563.718} C_VEL
LIN {X 0,Y 474.973,Z 916.111,A -85,B 0,C 180,E1 9563.261,E2 9563.261} C_VEL
LIN {X 0,Y 478.058,Z 887.73,A -85,B 0,C 180,E1 9562.773,E2 9562.773} C_VEL
LIN {X 0,Y 495.785,Z 668.628,A -85,B 0,C 180,E1 9559.392,E2 9559.392} C_VEL
LIN {X 0,Y 498.808,Z 632.26,A -85,B 0,C 180,E1 9558.828,E2 9558.828} C_VEL
LIN {X 0,Y 495.308,Z 626.175,A -85,B 0,C 180,E1 9557.323,E2 9557.323} C_VEL
LIN {X 0,Y 490.041,Z 617.773,A -85,B 0,C 180,E1 9554.777,E2 9554.777} C_VEL
LIN {X 0,Y 487.07,Z 613.18,A -85,B 0,C 180,E1 9553.111,E2 9553.111} C_VEL
LIN {X 0,Y 484.797,Z 609.598,A -85,B 0,C 180,E1 9551.661,E2 9551.661} C_VEL
LIN {X 0,Y 482.263,Z 605.697,A -85,B 0,C 180,E1 9549.789,E2 9549.789} C_VEL
LIN {X 0,Y 479.301,Z 600.983,A -85,B 0,C 180,E1 9546.95,E2 9546.95} C_VEL
LIN {X 0,Y 476.88,Z 597.34,A -85,B 0,C 180,E1 9543.125,E2 9543.125} C_VEL
LIN {X 0,Y 476.553,Z 595.737,A -85,B 0,C 180,E1 9541.683,E2 9541.683} C_VEL
LIN {X 0,Y 476.618,Z 595.851,A -85,B 0,C 180,E1 9537.836,E2 9537.836} C_VEL
LIN {X 0,Y 478.15,Z 599.846,A -85,B 0,C 180,E1 9534.239,E2 9534.239} C_VEL
LIN {X 0,Y 479.662,Z 601.488,A -85,B 0,C 180,E1 9532.454,E2 9532.454} C_VEL
LIN {X 0,Y 482.631,Z 606.035,A -85,B 0,C 180,E1 9529.737,E2 9529.737} C_VEL
LIN {X 0,Y 486.482,Z 612.168,A -85,B 0,C 180,E1 9527.054,E2 9527.054} C_VEL
LIN {X 0,Y 489.908,Z 617.499,A -85,B 0,C 180,E1 9525.098,E2 9525.098} C_VEL
LIN {X 0,Y 495.029,Z 625.65,A -85,B 0,C 180,E1 9522.606,E2 9522.606} C_VEL
LIN {X 0,Y 498.753,Z 631.929,A -85,B 0,C 180,E1 9521.005,E2 9521.005} C_VEL
LIN {X 0,Y 481.179,Z 846.809,A -85,B 0,C 180,E1 9517.695,E2 9517.695} C_VEL
LIN {X 0,Y 476.606,Z 900.616,A -85,B 0,C 180,E1 9516.844,E2 9516.844} C_VEL
LIN {X 0,Y 472.386,Z 930.232,A -85,B 0,C 180,E1 9516.268,E2 9516.268} C_VEL
LIN {X 0,Y 468.062,Z 952.866,A -85,B 0,C 180,E1 9515.698,E2 9515.698} C_VEL
LIN {X 0,Y 463.413,Z 973.257,A -85,B 0,C 180,E1 9515.064,E2 9515.064} C_VEL
LIN {X 0,Y 458.186,Z 993.061,A -85,B 0,C 180,E1 9514.33,E2 9514.33} C_VEL
LIN {X 0,Y 451.805,Z 1014.337,A -85,B 0,C 180,E1 9513.395,E2 9513.395} C_VEL
LIN {X 0,Y 442.633,Z 1041.033,A -85,B 0,C 180,E1 9511.974,E2 9511.974} C_VEL
LIN {X 0,Y 434.374,Z 1062.245,A -85,B 0,C 180,E1 9510.61,E2 9510.61} C_VEL
LIN {X 0,Y 426.543,Z 1080.744,A -85,B 0,C 180,E1 9509.223,E2 9509.223} C_VEL
LIN {X 0,Y 418.625,Z 1098.096,A -85,B 0,C 180,E1 9507.732,E2 9507.732} C_VEL
LIN {X 0,Y 408.908,Z 1118.071,A -85,B 0,C 180,E1 9505.744,E2 9505.744} C_VEL
LIN {X 0,Y 397.984,Z 1138.881,A -85,B 0,C 180,E1 9503.272,E2 9503.272} C_VEL
LIN {X 0,Y 389.077,Z 1154.979,A -85,B 0,C 180,E1 9501.026,E2 9501.026} C_VEL
LIN {X 0,Y 380.744,Z 1169.534,A -85,B 0,C 180,E1 9498.687,E2 9498.687} C_VEL
LIN {X 0,Y 371.904,Z 1184.637,A -85,B 0,C 180,E1 9495.881,E2 9495.881} C_VEL
LIN {X 0,Y 361.519,Z 1202.064,A -85,B 0,C 180,E1 9492.018,E2 9492.018} C_VEL
LIN {X 0,Y 354.247,Z 1214.232,A -85,B 0,C 180,E1 9488.804,E2 9488.804} C_VEL
LIN {X 0,Y 348.2,Z 1224.576,A -85,B 0,C 180,E1 9485.643,E2 9485.643} C_VEL
LIN {X 0,Y 342.855,Z 1234.157,A -85,B 0,C 180,E1 9482.248,E2 9482.248} C_VEL
LIN {X 0,Y 337.466,Z 1244.553,A -85,B 0,C 180,E1 9477.918,E2 9477.918} C_VEL
LIN {X 0,Y 333.318,Z 1253.393,A -85,B 0,C 180,E1 9473.331,E2 9473.331} C_VEL
LIN {X 0,Y 330.898,Z 1259.486,A -85,B 0,C 180,E1 9469.474,E2 9469.474} C_VEL
LIN {X 0,Y 329.396,Z 1264.148,A -85,B 0,C 180,E1 9465.859,E2 9465.859} C_VEL
LIN {X 0,Y 328.54,Z 1267.78,A -85,B 0,C 180,E1 9462.305,E2 9462.305} C_VEL
LIN {X 0,Y 328.104,Z 1270.485,A -85,B 0,C 180,E1 9458.769,E2 9458.769} C_VEL
LIN {X 0,Y 327.953,Z 1272.217,A -85,B 0,C 180,E1 9455.428,E2 9455.428} C_VEL
LIN {X 0,Y 327.914,Z 1273.143,A -85,B 0,C 180,E1 9452.102,E2 9452.102} C_VEL
LIN {X 0,Y 327.891,Z 1273.27,A -85,B 0,C 180,E1 9448.782,E2 9448.782} C_VEL
LIN {X 0,Y 327.935,Z 1272.528,A -85,B 0,C 180,E1 9445.283,E2 9445.283} C_VEL
LIN {X 0,Y 328.048,Z 1270.892,A -85,B 0,C 180,E1 9441.769,E2 9441.769} C_VEL
LIN {X 0,Y 328.459,Z 1268.193,A -85,B 0,C 180,E1 9438.059,E2 9438.059} C_VEL
LIN {X 0,Y 329.252,Z 1264.681,A -85,B 0,C 180,E1 9434.506,E2 9434.506} C_VEL
LIN {X 0,Y 330.744,Z 1259.967,A -85,B 0,C 180,E1 9430.766,E2 9430.766} C_VEL
LIN {X 0,Y 332.975,Z 1254.175,A -85,B 0,C 180,E1 9427.029,E2 9427.029} C_VEL
LIN {X 0,Y 336.095,Z 1247.262,A -85,B 0,C 180,E1 9423.313,E2 9423.313} C_VEL
LIN {X 0,Y 341.246,Z 1237.261,A -85,B 0,C 180,E1 9418.826,E2 9418.826} C_VEL
LIN {X 0,Y 347.514,Z 1225.841,A -85,B 0,C 180,E1 9414.675,E2 9414.675} C_VEL
LIN {X 0,Y 353.771,Z 1215.076,A -85,B 0,C 180,E1 9411.337,E2 9411.337} C_VEL
LIN {X 0,Y 360.728,Z 1203.403,A -85,B 0,C 180,E1 9408.214,E2 9408.214} C_VEL
LIN {X 0,Y 364.154,Z 1197.772,A -85,B 0,C 180,E1 9406.848,E2 9406.848} C_VEL
LIN {X 0,Y 365.73,Z 1193.807,A -85,B 0,C 180,E1 9405.835,E2 9405.835} C_VEL
LIN {X 0,Y 367.21,Z 1184.17,A -85,B 0,C 180,E1 9403.081,E2 9403.081} C_VEL
LIN {X 0,Y 369.162,Z 1179.862,A -85,B 0,C 180,E1 9402.117,E2 9402.117} C_VEL
LIN {X 0,Y 380.244,Z 1161.559,A -85,B 0,C 180,E1 9398.9,E2 9398.9} C_VEL
LIN {X 0,Y 390.303,Z 1144.053,A -85,B 0,C 180,E1 9396.334,E2 9396.334} C_VEL
LIN {X 0,Y 399.11,Z 1128.063,A -85,B 0,C 180,E1 9394.312,E2 9394.312} C_VEL
LIN {X 0,Y 407.869,Z 1111.31,A -85,B 0,C 180,E1 9392.472,E2 9392.472} C_VEL
LIN {X 0,Y 417.446,Z 1091.854,A -85,B 0,C 180,E1 9390.63,E2 9390.63} C_VEL
LIN {X 0,Y 428.49,Z 1067.222,A -85,B 0,C 180,E1 9388.682,E2 9388.682} C_VEL
LIN {X 0,Y 436.707,Z 1046.999,A -85,B 0,C 180,E1 9387.345,E2 9387.345} C_VEL
LIN {X 0,Y 444.064,Z 1027.041,A -85,B 0,C 180,E1 9386.209,E2 9386.209} C_VEL
LIN {X 0,Y 451.606,Z 1004.283,A -85,B 0,C 180,E1 9385.116,E2 9385.116} C_VEL
LIN {X 0,Y 459.118,Z 977.704,A -85,B 0,C 180,E1 9384.075,E2 9384.075} C_VEL
LIN {X 0,Y 464.467,Z 955.172,A -85,B 0,C 180,E1 9383.363,E2 9383.363} C_VEL
LIN {X 0,Y 468.726,Z 933.732,A -85,B 0,C 180,E1 9382.813,E2 9382.813} C_VEL
LIN {X 0,Y 472.352,Z 910.961,A -85,B 0,C 180,E1 9382.349,E2 9382.349} C_VEL
LIN {X 0,Y 475.754,Z 878.662,A -85,B 0,C 180,E1 9381.808,E2 9381.808} C_VEL
LIN {X 0,Y 494.019,Z 659.359,A -85,B 0,C 180,E1 9378.441,E2 9378.441} C_VEL
LIN {X 0,Y 495.882,Z 637.248,A -85,B 0,C 180,E1 9378.091,E2 9378.091} C_VEL
LIN {X 0,Y 490.666,Z 628.676,A -85,B 0,C 180,E1 9375.665,E2 9375.665} C_VEL
LIN {X 0,Y 486.473,Z 621.922,A -85,B 0,C 180,E1 9373.37,E2 9373.37} C_VEL
LIN {X 0,Y 483.588,Z 617.361,A -85,B 0,C 180,E1 9371.509,E2 9371.509} C_VEL
LIN {X 0,Y 481.206,Z 613.596,A -85,B 0,C 180,E1 9369.69,E2 9369.69} C_VEL
LIN {X 0,Y 478.342,Z 608.945,A -85,B 0,C 180,E1 9366.843,E2 9366.843} C_VEL
LIN {X 0,Y 476.014,Z 605.338,A -85,B 0,C 180,E1 9362.89,E2 9362.89} C_VEL
LIN {X 0,Y 475.746,Z 603.722,A -85,B 0,C 180,E1 9361.325,E2 9361.325} C_VEL
LIN {X 0,Y 475.795,Z 603.925,A -85,B 0,C 180,E1 9358.435,E2 9358.435} C_VEL
LIN {X 0,Y 477.285,Z 607.907,A -85,B 0,C 180,E1 9354.591,E2 9354.591} C_VEL
LIN {X 0,Y 478.69,Z 609.486,A -85,B 0,C 180,E1 9352.861,E2 9352.861} C_VEL
LIN {X 0,Y 481.488,Z 613.924,A -85,B 0,C 180,E1 9350.195,E2 9350.195} C_VEL
LIN {X 0,Y 485.047,Z 619.692,A -85,B 0,C 180,E1 9347.62,E2 9347.62} C_VEL
LIN {X 0,Y 488.572,Z 625.295,A -85,B 0,C 180,E1 9345.541,E2 9345.541} C_VEL
LIN {X 0,Y 493.83,Z 633.872,A -85,B 0,C 180,E1 9342.927,E2 9342.927} C_VEL
LIN {X 0,Y 495.964,Z 637.679,A -85,B 0,C 180,E1 9341.969,E2 9341.969} C_VEL
LIN {X 0,Y 477.897,Z 853.671,A -85,B 0,C 180,E1 9338.652,E2 9338.652} C_VEL
LIN {X 0,Y 473.403,Z 905.101,A -85,B 0,C 180,E1 9337.839,E2 9337.839} C_VEL
LIN {X 0,Y 469.094,Z 934.504,A -85,B 0,C 180,E1 9337.277,E2 9337.277} C_VEL
LIN {X 0,Y 464.724,Z 956.787,A -85,B 0,C 180,E1 9336.734,E2 9336.734} C_VEL
LIN {X 0,Y 459.814,Z 977.732,A -85,B 0,C 180,E1 9336.105,E2 9336.105} C_VEL
LIN {X 0,Y 454.257,Z 998.207,A -85,B 0,C 180,E1 9335.363,E2 9335.363} C_VEL
LIN {X 0,Y 446.76,Z 1022.427,A -85,B 0,C 180,E1 9334.308,E2 9334.308} C_VEL
LIN {X 0,Y 437.683,Z 1047.615,A -85,B 0,C 180,E1 9332.96,E2 9332.96} C_VEL
LIN {X 0,Y 429.795,Z 1067.385,A -85,B 0,C 180,E1 9331.696,E2 9331.696} C_VEL
LIN {X 0,Y 422.058,Z 1085.208,A -85,B 0,C 180,E1 9330.382,E2 9330.382} C_VEL
LIN {X 0,Y 413.572,Z 1103.361,A -85,B 0,C 180,E1 9328.843,E2 9328.843} C_VEL
LIN {X 0,Y 402.664,Z 1125.245,A -85,B 0,C 180,E1 9326.666,E2 9326.666} C_VEL
LIN {X 0,Y 391.736,Z 1145.358,A -85,B 0,C 180,E1 9324.249,E2 9324.249} C_VEL
LIN {X 0,Y 382.7,Z 1161.277,A -85,B 0,C 180,E1 9322.019,E2 9322.019} C_VEL
LIN {X 0,Y 374.014,Z 1176.079,A -85,B 0,C 180,E1 9319.624,E2 9319.624} C_VEL
LIN {X 0,Y 363.717,Z 1193.318,A -85,B 0,C 180,E1 9316.368,E2 9316.368} C_VEL
LIN {X 0,Y 353.927,Z 1209.192,A -85,B 0,C 180,E1 9312.732,E2 9312.732} C_VEL
LIN {X 0,Y 346.749,Z 1220.946,A -85,B 0,C 180,E1 9309.581,E2 9309.581} C_VEL
LIN {X 0,Y 340.243,Z 1231.835,A -85,B 0,C 180,E1 9306.198,E2 9306.198} C_VEL
LIN {X 0,Y 333.56,Z 1243.766,A -85,B 0,C 180,E1 9301.835,E2 9301.835} C_VEL
LIN {X 0,Y 328.353,Z 1253.656,A -85,B 0,C 180,E1 9297.368,E2 9297.368} C_VEL
LIN {X 0,Y 325.112,Z 1260.718,A -85,B 0,C 180,E1 9293.56,E2 9293.56} C_VEL
LIN {X 0,Y 322.759,Z 1266.646,A -85,B 0,C 180,E1 9289.729,E2 9289.729} C_VEL
LIN {X 0,Y 321.286,Z 1271.273,A -85,B 0,C 180,E1 9286.074,E2 9286.074} C_VEL
LIN {X 0,Y 320.447,Z 1274.955,A -85,B 0,C 180,E1 9282.404,E2 9282.404} C_VEL
LIN {X 0,Y 320.05,Z 1277.649,A -85,B 0,C 180,E1 9278.8,E2 9278.8} C_VEL
LIN {X 0,Y 319.93,Z 1279.367,A -85,B 0,C 180,E1 9275.375,E2 9275.375} C_VEL
LIN {X 0,Y 319.911,Z 1280.258,A -85,B 0,C 180,E1 9271.965,E2 9271.965} C_VEL
LIN {X 0,Y 319.902,Z 1280.324,A -85,B 0,C 180,E1 9268.562,E2 9268.562} C_VEL
LIN {X 0,Y 319.923,Z 1279.566,A -85,B 0,C 180,E1 9265.154,E2 9265.154} C_VEL
LIN {X 0,Y 320.019,Z 1277.866,A -85,B 0,C 180,E1 9261.551,E2 9261.551} C_VEL
LIN {X 0,Y 320.421,Z 1275.076,A -85,B 0,C 180,E1 9257.744,E2 9257.744} C_VEL
LIN {X 0,Y 321.23,Z 1271.458,A -85,B 0,C 180,E1 9254.098,E2 9254.098} C_VEL
LIN {X 0,Y 322.709,Z 1266.781,A -85,B 0,C 180,E1 9250.378,E2 9250.378} C_VEL
LIN {X 0,Y 324.984,Z 1260.986,A -85,B 0,C 180,E1 9246.611,E2 9246.611} C_VEL
LIN {X 0,Y 328.18,Z 1253.966,A -85,B 0,C 180,E1 9242.801,E2 9242.801} C_VEL
LIN {X 0,Y 333.328,Z 1244.13,A -85,B 0,C 180,E1 9238.331,E2 9238.331} C_VEL
LIN {X 0,Y 339.958,Z 1232.29,A -85,B 0,C 180,E1 9233.964,E2 9233.964} C_VEL
LIN {X 0,Y 346.412,Z 1221.448,A -85,B 0,C 180,E1 9230.575,E2 9230.575} C_VEL
LIN {X 0,Y 353.454,Z 1209.888,A -85,B 0,C 180,E1 9227.456,E2 9227.456} C_VEL
LIN {X 0,Y 361.796,Z 1196.278,A -85,B 0,C 180,E1 9224.288,E2 9224.288} C_VEL
LIN {X 0,Y 373.038,Z 1177.642,A -85,B 0,C 180,E1 9220.66,E2 9220.66} C_VEL
LIN {X 0,Y 382.067,Z 1162.261,A -85,B 0,C 180,E1 9218.143,E2 9218.143} C_VEL
LIN {X 0,Y 390.903,Z 1146.714,A -85,B 0,C 180,E1 9215.942,E2 9215.942} C_VEL
LIN {X 0,Y 399.966,Z 1130.067,A -85,B 0,C 180,E1 9213.9,E2 9213.9} C_VEL
LIN {X 0,Y 410.582,Z 1109.513,A -85,B 0,C 180,E1 9211.737,E2 9211.737} C_VEL
LIN {X 0,Y 420.763,Z 1087.873,A -85,B 0,C 180,E1 9209.842,E2 9209.842} C_VEL
LIN {X 0,Y 428.789,Z 1069.512,A -85,B 0,C 180,E1 9208.46,E2 9208.46} C_VEL
LIN {X 0,Y 436.355,Z 1050.753,A -85,B 0,C 180,E1 9207.238,E2 9207.238} C_VEL
LIN {X 0,Y 443.411,Z 1031.638,A -85,B 0,C 180,E1 9206.168,E2 9206.168} C_VEL
LIN {X 0,Y 450.256,Z 1011.084,A -85,B 0,C 180,E1 9205.182,E2 9205.182} C_VEL
LIN {X 0,Y 457.987,Z 984.544,A -85,B 0,C 180,E1 9204.132,E2 9204.132} C_VEL
LIN {X 0,Y 463.879,Z 960.058,A -85,B 0,C 180,E1 9203.362,E2 9203.362} C_VEL
LIN {X 0,Y 468.208,Z 938.608,A -85,B 0,C 180,E1 9202.822,E2 9202.822} C_VEL
LIN {X 0,Y 471.785,Z 916.496,A -85,B 0,C 180,E1 9202.373,E2 9202.373} C_VEL
LIN {X 0,Y 474.898,Z 888.919,A -85,B 0,C 180,E1 9201.899,E2 9201.899} C_VEL
LIN {X 0,Y 493.057,Z 669.854,A -85,B 0,C 180,E1 9198.531,E2 9198.531} C_VEL
LIN {X 0,Y 495.761,Z 637.364,A -85,B 0,C 180,E1 9198.007,E2 9198.007} C_VEL
LIN {X 0,Y 491.869,Z 630.734,A -85,B 0,C 180,E1 9196.231,E2 9196.231} C_VEL
LIN {X 0,Y 486.877,Z 622.582,A -85,B 0,C 180,E1 9193.6,E2 9193.6} C_VEL
LIN {X 0,Y 483.383,Z 617.167,A -85,B 0,C 180,E1 9191.393,E2 9191.393} C_VEL
LIN {X 0,Y 481.138,Z 613.58,A -85,B 0,C 180,E1 9189.691,E2 9189.691} C_VEL
LIN {X 0,Y 478.218,Z 608.866,A -85,B 0,C 180,E1 9186.845,E2 9186.845} C_VEL
LIN {X 0,Y 475.859,Z 605.22,A -85,B 0,C 180,E1 9183.011,E2 9183.011} C_VEL
LIN {X 0,Y 475.549,Z 603.67,A -85,B 0,C 180,E1 9181.566,E2 9181.566} C_VEL
LIN {X 0,Y 475.63,Z 603.905,A -85,B 0,C 180,E1 9177.831,E2 9177.831} C_VEL
LIN {X 0,Y 477.351,Z 608.04,A -85,B 0,C 180,E1 9173.988,E2 9173.988} C_VEL
LIN {X 0,Y 478.567,Z 609.42,A -85,B 0,C 180,E1 9172.557,E2 9172.557} C_VEL
LIN {X 0,Y 481.929,Z 614.806,A -85,B 0,C 180,E1 9169.48,E2 9169.48} C_VEL
LIN {X 0,Y 485.119,Z 619.868,A -85,B 0,C 180,E1 9167.259,E2 9167.259} C_VEL
LIN {X 0,Y 488.485,Z 625.213,A -85,B 0,C 180,E1 9165.296,E2 9165.296} C_VEL
LIN {X 0,Y 494.025,Z 634.224,A -85,B 0,C 180,E1 9162.569,E2 9162.569} C_VEL
LIN {X 0,Y 495.739,Z 637.392,A -85,B 0,C 180,E1 9161.8,E2 9161.8} C_VEL
LIN {X 0,Y 477.642,Z 853.658,A -85,B 0,C 180,E1 9158.481,E2 9158.481} C_VEL
LIN {X 0,Y 473.368,Z 902.117,A -85,B 0,C 180,E1 9157.713,E2 9157.713} C_VEL
LIN {X 0,Y 469.135,Z 930.763,A -85,B 0,C 180,E1 9157.156,E2 9157.156} C_VEL
LIN {X 0,Y 464.762,Z 953.182,A -85,B 0,C 180,E1 9156.596,E2 9156.596} C_VEL
LIN {X 0,Y 459.887,Z 974.094,A -85,B 0,C 180,E1 9155.949,E2 9155.949} C_VEL
LIN {X 0,Y 454.379,Z 994.44,A -85,B 0,C 180,E1 9155.196,E2 9155.196} C_VEL
LIN {X 0,Y 446.816,Z 1018.945,A -85,B 0,C 180,E1 9154.108,E2 9154.108} C_VEL
LIN {X 0,Y 437.983,Z 1043.394,A -85,B 0,C 180,E1 9152.776,E2 9152.776} C_VEL
LIN {X 0,Y 430.083,Z 1063.149,A -85,B 0,C 180,E1 9151.501,E2 9151.501} C_VEL
LIN {X 0,Y 422.077,Z 1081.571,A -85,B 0,C 180,E1 9150.12,E2 9150.12} C_VEL
LIN {X 0,Y 413.653,Z 1099.521,A -85,B 0,C 180,E1 9148.573,E2 9148.573} C_VEL
LIN {X 0,Y 402.502,Z 1121.661,A -85,B 0,C 180,E1 9146.329,E2 9146.329} C_VEL
LIN {X 0,Y 392.217,Z 1140.488,A -85,B 0,C 180,E1 9144.042,E2 9144.042} C_VEL
LIN {X 0,Y 383.62,Z 1155.534,A -85,B 0,C 180,E1 9141.923,E2 9141.923} C_VEL
LIN {X 0,Y 374.781,Z 1170.469,A -85,B 0,C 180,E1 9139.499,E2 9139.499} C_VEL
LIN {X 0,Y 365.217,Z 1186.263,A -85,B 0,C 180,E1 9136.515,E2 9136.515} C_VEL
LIN {X 0,Y 354.937,Z 1202.789,A -85,B 0,C 180,E1 9132.763,E2 9132.763} C_VEL
LIN {X 0,Y 347.403,Z 1214.895,A -85,B 0,C 180,E1 9129.504,E2 9129.504} C_VEL
LIN {X 0,Y 341.099,Z 1225.215,A -85,B 0,C 180,E1 9126.28,E2 9126.28} C_VEL
LIN {X 0,Y 335.315,Z 1235.133,A -85,B 0,C 180,E1 9122.669,E2 9122.669} C_VEL
LIN {X 0,Y 329.339,Z 1246.094,A -85,B 0,C 180,E1 9117.88,E2 9117.88} C_VEL
LIN {X 0,Y 325.585,Z 1253.785,A -85,B 0,C 180,E1 9113.727,E2 9113.727} C_VEL
LIN {X 0,Y 323.107,Z 1259.654,A -85,B 0,C 180,E1 9109.906,E2 9109.906} C_VEL
LIN {X 0,Y 321.532,Z 1264.239,A -85,B 0,C 180,E1 9106.258,E2 9106.258} C_VEL
LIN {X 0,Y 320.599,Z 1267.869,A -85,B 0,C 180,E1 9102.615,E2 9102.615} C_VEL
LIN {X 0,Y 320.125,Z 1270.574,A -85,B 0,C 180,E1 9098.99,E2 9098.99} C_VEL
LIN {X 0,Y 319.959,Z 1272.305,A -85,B 0,C 180,E1 9095.564,E2 9095.564} C_VEL
LIN {X 0,Y 319.914,Z 1273.231,A -85,B 0,C 180,E1 9092.154,E2 9092.154} C_VEL
LIN {X 0,Y 319.893,Z 1273.357,A -85,B 0,C 180,E1 9088.751,E2 9088.751} C_VEL
LIN {X 0,Y 319.938,Z 1272.615,A -85,B 0,C 180,E1 9085.165,E2 9085.165} C_VEL
LIN {X 0,Y 320.066,Z 1270.98,A -85,B 0,C 180,E1 9081.562,E2 9081.562} C_VEL
LIN {X 0,Y 320.512,Z 1268.282,A -85,B 0,C 180,E1 9077.758,E2 9077.758} C_VEL
LIN {X 0,Y 321.407,Z 1264.649,A -85,B 0,C 180,E1 9074.007,E2 9074.007} C_VEL
LIN {X 0,Y 322.996,Z 1259.988,A -85,B 0,C 180,E1 9070.235,E2 9070.235} C_VEL
LIN {X 0,Y 325.372,Z 1254.264,A -85,B 0,C 180,E1 9066.46,E2 9066.46} C_VEL
LIN {X 0,Y 328.677,Z 1247.351,A -85,B 0,C 180,E1 9062.661,E2 9062.661} C_VEL
LIN {X 0,Y 333.953,Z 1237.654,A -85,B 0,C 180,E1 9058.207,E2 9058.207} C_VEL
LIN {X 0,Y 340.701,Z 1225.931,A -85,B 0,C 180,E1 9053.859,E2 9053.859} C_VEL
LIN {X 0,Y 347.237,Z 1215.211,A -85,B 0,C 180,E1 9050.486,E2 9050.486} C_VEL
LIN {X 0,Y 354.352,Z 1203.77,A -85,B 0,C 180,E1 9047.382,E2 9047.382} C_VEL
LIN {X 0,Y 363.672,Z 1188.897,A -85,B 0,C 180,E1 9043.926,E2 9043.926} C_VEL
LIN {X 0,Y 369.162,Z 1179.862,A -85,B 0,C 180,E1 9042.117,E2 9042.117} C_VEL
LIN {X 0,Y 371.196,Z 1175.568,A -85,B 0,C 180,E1 9041.17,E2 9041.17} C_VEL
LIN {X 0,Y 373.967,Z 1164.32,A -85,B 0,C 180,E1 9038.431,E2 9038.431} C_VEL
LIN {X 0,Y 375.903,Z 1160.216,A -85,B 0,C 180,E1 9037.687,E2 9037.687} C_VEL
LIN {X 0,Y 385.726,Z 1143.636,A -85,B 0,C 180,E1 9035.27,E2 9035.27} C_VEL
LIN {X 0,Y 394.665,Z 1127.861,A -85,B 0,C 180,E1 9033.285,E2 9033.285} C_VEL
LIN {X 0,Y 403.664,Z 1111.09,A -85,B 0,C 180,E1 9031.453,E2 9031.453} C_VEL
LIN {X 0,Y 414.131,Z 1090.33,A -85,B 0,C 180,E1 9029.508,E2 9029.508} C_VEL
LIN {X 0,Y 424.625,Z 1067.306,A -85,B 0,C 180,E1 9027.714,E2 9027.714} C_VEL
LIN {X 0,Y 433.019,Z 1047.082,A -85,B 0,C 180,E1 9026.385,E2 9026.385} C_VEL
LIN {X 0,Y 440.567,Z 1027.039,A -85,B 0,C 180,E1 9025.257,E2 9025.257} C_VEL
LIN {X 0,Y 448.228,Z 1004.364,A -85,B 0,C 180,E1 9024.179,E2 9024.179} C_VEL
LIN {X 0,Y 455.886,Z 977.782,A -85,B 0,C 180,E1 9023.15,E2 9023.15} C_VEL
LIN {X 0,Y 461.334,Z 955.249,A -85,B 0,C 180,E1 9022.446,E2 9022.446} C_VEL
LIN {X 0,Y 465.671,Z 933.806,A -85,B 0,C 180,E1 9021.903,E2 9021.903} C_VEL
LIN {X 0,Y 469.359,Z 911.032,A -85,B 0,C 180,E1 9021.443,E2 9021.443} C_VEL
LIN {X 0,Y 472.834,Z 878.689,A -85,B 0,C 180,E1 9020.905,E2 9020.905} C_VEL
LIN {X 0,Y 491.514,Z 659.69,A -85,B 0,C 180,E1 9017.557,E2 9017.557} C_VEL
LIN {X 0,Y 492.983,Z 642.609,A -85,B 0,C 180,E1 9017.286,E2 9017.286} C_VEL
LIN {X 0,Y 487.284,Z 633.197,A -85,B 0,C 180,E1 9014.437,E2 9014.437} C_VEL
LIN {X 0,Y 483.893,Z 627.698,A -85,B 0,C 180,E1 9012.41,E2 9012.41} C_VEL
LIN {X 0,Y 481.702,Z 624.192,A -85,B 0,C 180,E1 9010.888,E2 9010.888} C_VEL
LIN {X 0,Y 479.94,Z 621.316,A -85,B 0,C 180,E1 9009.473,E2 9009.473} C_VEL
LIN {X 0,Y 477.263,Z 616.829,A -85,B 0,C 180,E1 9006.738,E2 9006.738} C_VEL
LIN {X 0,Y 474.999,Z 613.218,A -85,B 0,C 180,E1 9002.775,E2 9002.775} C_VEL
LIN {X 0,Y 474.751,Z 611.658,A -85,B 0,C 180,E1 9001.207,E2 9001.207} C_VEL
LIN {X 0,Y 474.81,Z 611.945,A -85,B 0,C 180,E1 8998.431,E2 8998.431} C_VEL
LIN {X 0,Y 476.309,Z 615.89,A -85,B 0,C 180,E1 8994.579,E2 8994.579} C_VEL
LIN {X 0,Y 477.6,Z 617.415,A -85,B 0,C 180,E1 8992.965,E2 8992.965} C_VEL
LIN {X 0,Y 480.858,Z 622.724,A -85,B 0,C 180,E1 8989.88,E2 8989.88} C_VEL
LIN {X 0,Y 483.871,Z 627.702,A -85,B 0,C 180,E1 8987.711,E2 8987.711} C_VEL
LIN {X 0,Y 487.261,Z 633.172,A -85,B 0,C 180,E1 8985.684,E2 8985.684} C_VEL
LIN {X 0,Y 493.016,Z 642.695,A -85,B 0,C 180,E1 8982.807,E2 8982.807} C_VEL
LIN {X 0,Y 483.012,Z 759.032,A -85,B 0,C 180,E1 8981.005,E2 8981.005} C_VEL
LIN {X 0,Y 470.845,Z 901.046,A -85,B 0,C 180,E1 8978.811,E2 8978.811} C_VEL
LIN {X 0,Y 467.222,Z 928.057,A -85,B 0,C 180,E1 8978.324,E2 8978.324} C_VEL
LIN {X 0,Y 462.012,Z 954.864,A -85,B 0,C 180,E1 8977.703,E2 8977.703} C_VEL
LIN {X 0,Y 456.963,Z 976.251,A -85,B 0,C 180,E1 8977.077,E2 8977.077} C_VEL
LIN {X 0,Y 451.428,Z 996.437,A -85,B 0,C 180,E1 8976.365,E2 8976.365} C_VEL
LIN {X 0,Y 444.99,Z 1017.107,A -85,B 0,C 180,E1 8975.495,E2 8975.495} C_VEL
LIN {X 0,Y 436.249,Z 1041.984,A -85,B 0,C 180,E1 8974.244,E2 8974.244} C_VEL
LIN {X 0,Y 426.672,Z 1065.673,A -85,B 0,C 180,E1 8972.777,E2 8972.777} C_VEL
LIN {X 0,Y 418.384,Z 1084.384,A -85,B 0,C 180,E1 8971.423,E2 8971.423} C_VEL
LIN {X 0,Y 409.684,Z 1102.604,A -85,B 0,C 180,E1 8969.893,E2 8969.893} C_VEL
LIN {X 0,Y 399.628,Z 1122.302,A -85,B 0,C 180,E1 8967.965,E2 8967.965} C_VEL
LIN {X 0,Y 387.51,Z 1144.252,A -85,B 0,C 180,E1 8965.386,E2 8965.386} C_VEL
LIN {X 0,Y 377.855,Z 1160.781,A -85,B 0,C 180,E1 8963.08,E2 8963.08} C_VEL
LIN {X 0,Y 368.638,Z 1175.99,A -85,B 0,C 180,E1 8960.616,E2 8960.616} C_VEL
LIN {X 0,Y 358.274,Z 1192.706,A -85,B 0,C 180,E1 8957.448,E2 8957.448} C_VEL
LIN {X 0,Y 348.105,Z 1208.61,A -85,B 0,C 180,E1 8953.799,E2 8953.799} C_VEL
LIN {X 0,Y 340.669,Z 1220.279,A -85,B 0,C 180,E1 8950.653,E2 8950.653} C_VEL
LIN {X 0,Y 333.814,Z 1231.226,A -85,B 0,C 180,E1 8947.225,E2 8947.225} C_VEL
LIN {X 0,Y 327.48,Z 1241.834,A -85,B 0,C 180,E1 8943.331,E2 8943.331} C_VEL
LIN {X 0,Y 321.347,Z 1252.852,A -85,B 0,C 180,E1 8938.422,E2 8938.422} C_VEL
LIN {X 0,Y 317.513,Z 1260.628,A -85,B 0,C 180,E1 8934.159,E2 8934.159} C_VEL
LIN {X 0,Y 314.997,Z 1266.556,A -85,B 0,C 180,E1 8930.236,E2 8930.236} C_VEL
LIN {X 0,Y 313.421,Z 1271.184,A -85,B 0,C 180,E1 8926.489,E2 8926.489} C_VEL
LIN {X 0,Y 312.474,Z 1274.988,A -85,B 0,C 180,E1 8922.584,E2 8922.584} C_VEL
LIN {X 0,Y 312.052,Z 1277.676,A -85,B 0,C 180,E1 8918.842,E2 8918.842} C_VEL
LIN {X 0,Y 311.929,Z 1279.348,A -85,B 0,C 180,E1 8915.328,E2 8915.328} C_VEL
LIN {X 0,Y 311.912,Z 1280.17,A -85,B 0,C 180,E1 8912.015,E2 8912.015} C_VEL
LIN {X 0,Y 311.904,Z 1280.236,A -85,B 0,C 180,E1 8908.525,E2 8908.525} C_VEL
LIN {X 0,Y 311.924,Z 1279.478,A -85,B 0,C 180,E1 8905.03,E2 8905.03} C_VEL
LIN {X 0,Y 312.036,Z 1277.777,A -85,B 0,C 180,E1 8901.333,E2 8901.333} C_VEL
LIN {X 0,Y 312.44,Z 1275.149,A -85,B 0,C 180,E1 8897.614,E2 8897.614} C_VEL
LIN {X 0,Y 313.357,Z 1271.368,A -85,B 0,C 180,E1 8893.687,E2 8893.687} C_VEL
LIN {X 0,Y 314.905,Z 1266.782,A -85,B 0,C 180,E1 8889.94,E2 8889.94} C_VEL
LIN {X 0,Y 317.38,Z 1260.889,A -85,B 0,C 180,E1 8886.013,E2 8886.013} C_VEL
LIN {X 0,Y 320.968,Z 1253.517,A -85,B 0,C 180,E1 8881.935,E2 8881.935} C_VEL
LIN {X 0,Y 326.73,Z 1243.16,A -85,B 0,C 180,E1 8877.198,E2 8877.198} C_VEL
LIN {X 0,Y 333.507,Z 1231.677,A -85,B 0,C 180,E1 8872.938,E2 8872.938} C_VEL
LIN {X 0,Y 340.319,Z 1220.777,A -85,B 0,C 180,E1 8869.506,E2 8869.506} C_VEL
LIN {X 0,Y 348.12,Z 1208.515,A -85,B 0,C 180,E1 8866.191,E2 8866.191} C_VEL
LIN {X 0,Y 358.608,Z 1192.055,A -85,B 0,C 180,E1 8862.436,E2 8862.436} C_VEL
LIN {X 0,Y 368.656,Z 1175.849,A -85,B 0,C 180,E1 8859.373,E2 8859.373} C_VEL
LIN {X 0,Y 377.806,Z 1160.732,A -85,B 0,C 180,E1 8856.925,E2 8856.925} C_VEL
LIN {X 0,Y 387.235,Z 1144.583,A -85,B 0,C 180,E1 8854.67,E2 8854.67} C_VEL
LIN {X 0,Y 399.111,Z 1123.123,A -85,B 0,C 180,E1 8852.133,E2 8852.133} C_VEL
LIN {X 0,Y 409.376,Z 1103.016,A -85,B 0,C 180,E1 8850.156,E2 8850.156} C_VEL
LIN {X 0,Y 418.067,Z 1084.83,A -85,B 0,C 180,E1 8848.624,E2 8848.624} C_VEL
LIN {X 0,Y 425.992,Z 1066.977,A -85,B 0,C 180,E1 8847.322,E2 8847.322} C_VEL
LIN {X 0,Y 434.463,Z 1046.147,A -85,B 0,C 180,E1 8846.008,E2 8846.008} C_VEL
LIN {X 0,Y 444.276,Z 1018.918,A -85,B 0,C 180,E1 8844.596,E2 8844.596} C_VEL
LIN {X 0,Y 450.959,Z 997.598,A -85,B 0,C 180,E1 8843.688,E2 8843.688} C_VEL
LIN {X 0,Y 456.624,Z 977.036,A -85,B 0,C 180,E1 8842.956,E2 8842.956} C_VEL
LIN {X 0,Y 461.721,Z 955.551,A -85,B 0,C 180,E1 8842.323,E2 8842.323} C_VEL
LIN {X 0,Y 466.674,Z 930.327,A -85,B 0,C 180,E1 8841.73,E2 8841.73} C_VEL
LIN {X 0,Y 470.583,Z 902.173,A -85,B 0,C 180,E1 8841.214,E2 8841.214} C_VEL
LIN {X 0,Y 477.893,Z 817.593,A -85,B 0,C 180,E1 8839.898,E2 8839.898} C_VEL
LIN {X 0,Y 492.895,Z 642.618,A -85,B 0,C 180,E1 8837.213,E2 8837.213} C_VEL
LIN {X 0,Y 487.087,Z 633.02,A -85,B 0,C 180,E1 8834.32,E2 8834.32} C_VEL
LIN {X 0,Y 482.748,Z 625.79,A -85,B 0,C 180,E1 8831.651,E2 8831.651} C_VEL
LIN {X 0,Y 479.867,Z 621.299,A -85,B 0,C 180,E1 8829.475,E2 8829.475} C_VEL
LIN {X 0,Y 477.03,Z 616.658,A -85,B 0,C 180,E1 8826.62,E2 8826.62} C_VEL
LIN {X 0,Y 474.807,Z 612.949,A -85,B 0,C 180,E1 8822.776,E2 8822.776} C_VEL
LIN {X 0,Y 474.547,Z 611.606,A -85,B 0,C 180,E1 8821.449,E2 8821.449} C_VEL
LIN {X 0,Y 474.627,Z 611.789,A -85,B 0,C 180,E1 8817.948,E2 8817.948} C_VEL
LIN {X 0,Y 476.286,Z 615.92,A -85,B 0,C 180,E1 8814.096,E2 8814.096} C_VEL
LIN {X 0,Y 477.475,Z 617.348,A -85,B 0,C 180,E1 8812.661,E2 8812.661} C_VEL
LIN {X 0,Y 480.643,Z 622.497,A -85,B 0,C 180,E1 8809.694,E2 8809.694} C_VEL
LIN {X 0,Y 483.852,Z 627.721,A -85,B 0,C 180,E1 8807.407,E2 8807.407} C_VEL
LIN {X 0,Y 487.068,Z 632.925,A -85,B 0,C 180,E1 8805.496,E2 8805.496} C_VEL
LIN {X 0,Y 492.851,Z 642.488,A -85,B 0,C 180,E1 8802.611,E2 8802.611} C_VEL
LIN {X 0,Y 474.462,Z 857.331,A -85,B 0,C 180,E1 8799.327,E2 8799.327} C_VEL
LIN {X 0,Y 470.262,Z 903.404,A -85,B 0,C 180,E1 8798.598,E2 8798.598} C_VEL
LIN {X 0,Y 466.015,Z 931.202,A -85,B 0,C 180,E1 8798.058,E2 8798.058} C_VEL
LIN {X 0,Y 461.602,Z 953.39,A -85,B 0,C 180,E1 8797.509,E2 8797.509} C_VEL
LIN {X 0,Y 456.661,Z 974.192,A -85,B 0,C 180,E1 8796.873,E2 8796.873} C_VEL
LIN {X 0,Y 451.048,Z 994.537,A -85,B 0,C 180,E1 8796.128,E2 8796.128} C_VEL
LIN {X 0,Y 443.333,Z 1019.041,A -85,B 0,C 180,E1 8795.052,E2 8795.052} C_VEL
LIN {X 0,Y 434.316,Z 1043.49,A -85,B 0,C 180,E1 8793.732,E2 8793.732} C_VEL
LIN {X 0,Y 426.247,Z 1063.244,A -85,B 0,C 180,E1 8792.466,E2 8792.466} C_VEL
LIN {X 0,Y 418.199,Z 1081.345,A -85,B 0,C 180,E1 8791.12,E2 8791.12} C_VEL
LIN {X 0,Y 409.418,Z 1099.616,A -85,B 0,C 180,E1 8789.557,E2 8789.557} C_VEL
LIN {X 0,Y 397.83,Z 1122.012,A -85,B 0,C 180,E1 8787.291,E2 8787.291} C_VEL
LIN {X 0,Y 387.434,Z 1140.521,A -85,B 0,C 180,E1 8785.044,E2 8785.044} C_VEL
LIN {X 0,Y 378.134,Z 1156.304,A -85,B 0,C 180,E1 8782.813,E2 8782.813} C_VEL
LIN {X 0,Y 368.897,Z 1171.404,A -85,B 0,C 180,E1 8780.337,E2 8780.337} C_VEL
LIN {X 0,Y 358.109,Z 1188.606,A -85,B 0,C 180,E1 8777.019,E2 8777.019} C_VEL
LIN {X 0,Y 348.417,Z 1203.513,A -85,B 0,C 180,E1 8773.535,E2 8773.535} C_VEL
LIN {X 0,Y 340.983,Z 1214.989,A -85,B 0,C 180,E1 8770.399,E2 8770.399} C_VEL
LIN {X 0,Y 334.114,Z 1225.739,A -85,B 0,C 180,E1 8766.983,E2 8766.983} C_VEL
LIN {X 0,Y 327.257,Z 1237.046,A -85,B 0,C 180,E1 8762.742,E2 8762.742} C_VEL
LIN {X 0,Y 321.399,Z 1247.236,A -85,B 0,C 180,E1 8758.024,E2 8758.024} C_VEL
LIN {X 0,Y 317.866,Z 1254.176,A -85,B 0,C 180,E1 8754.142,E2 8754.142} C_VEL
LIN {X 0,Y 315.265,Z 1259.997,A -85,B 0,C 180,E1 8750.229,E2 8750.229} C_VEL
LIN {X 0,Y 313.612,Z 1264.533,A -85,B 0,C 180,E1 8746.489,E2 8746.489} C_VEL
LIN {X 0,Y 312.593,Z 1268.274,A -85,B 0,C 180,E1 8742.568,E2 8742.568} C_VEL
LIN {X 0,Y 312.092,Z 1270.999,A -85,B 0,C 180,E1 8738.665,E2 8738.665} C_VEL
LIN {X 0,Y 311.943,Z 1272.662,A -85,B 0,C 180,E1 8734.97,E2 8734.97} C_VEL
LIN {X 0,Y 311.901,Z 1273.431,A -85,B 0,C 180,E1 8731.291,E2 8731.291} C_VEL
LIN {X 0,Y 311.915,Z 1273.31,A -85,B 0,C 180,E1 8727.617,E2 8727.617} C_VEL
LIN {X 0,Y 311.974,Z 1272.301,A -85,B 0,C 180,E1 8723.934,E2 8723.934} C_VEL
LIN {X 0,Y 312.161,Z 1270.396,A -85,B 0,C 180,E1 8720.232,E2 8720.232} C_VEL
LIN {X 0,Y 312.8,Z 1267.424,A -85,B 0,C 180,E1 8716.323,E2 8716.323} C_VEL
LIN {X 0,Y 314.448,Z 1262.282,A -85,B 0,C 180,E1 8711.369,E2 8711.369} C_VEL
LIN {X 0,Y 317.216,Z 1255.553,A -85,B 0,C 180,E1 8706.606,E2 8706.606} C_VEL
LIN {X 0,Y 320.545,Z 1248.84,A -85,B 0,C 180,E1 8702.714,E2 8702.714} C_VEL
LIN {X 0,Y 324.687,Z 1241.359,A -85,B 0,C 180,E1 8699.058,E2 8699.058} C_VEL
LIN {X 0,Y 330.087,Z 1232.298,A -85,B 0,C 180,E1 8695.294,E2 8695.294} C_VEL
LIN {X 0,Y 337.972,Z 1219.855,A -85,B 0,C 180,E1 8690.947,E2 8690.947} C_VEL
LIN {X 0,Y 346.584,Z 1206.382,A -85,B 0,C 180,E1 8687.098,E2 8687.098} C_VEL
LIN {X 0,Y 354.696,Z 1193.86,A -85,B 0,C 180,E1 8684.05,E2 8684.05} C_VEL
LIN {X 0,Y 363.162,Z 1180.646,A -85,B 0,C 180,E1 8681.277,E2 8681.277} C_VEL
LIN {X 0,Y 373.989,Z 1163.448,A -85,B 0,C 180,E1 8678.194,E2 8678.194} C_VEL
LIN {X 0,Y 375.903,Z 1160.216,A -85,B 0,C 180,E1 8677.687,E2 8677.687} C_VEL
LIN {X 0,Y 378.117,Z 1155.481,A -85,B 0,C 180,E1 8676.824,E2 8676.824} C_VEL
LIN {X 0,Y 381.467,Z 1143.893,A -85,B 0,C 180,E1 8674.393,E2 8674.393} C_VEL
LIN {X 0,Y 383.936,Z 1138.774,A -85,B 0,C 180,E1 8673.59,E2 8673.59} C_VEL
LIN {X 0,Y 396.534,Z 1116.556,A -85,B 0,C 180,E1 8670.994,E2 8670.994} C_VEL
LIN {X 0,Y 406.411,Z 1097.733,A -85,B 0,C 180,E1 8669.157,E2 8669.157} C_VEL
LIN {X 0,Y 415.298,Z 1079.578,A -85,B 0,C 180,E1 8667.638,E2 8667.638} C_VEL
LIN {X 0,Y 423.731,Z 1060.915,A -85,B 0,C 180,E1 8666.287,E2 8666.287} C_VEL
LIN {X 0,Y 433.835,Z 1036.229,A -85,B 0,C 180,E1 8664.774,E2 8664.774} C_VEL
LIN {X 0,Y 441.966,Z 1013.469,A -85,B 0,C 180,E1 8663.63,E2 8663.63} C_VEL
LIN {X 0,Y 448.368,Z 993.316,A -85,B 0,C 180,E1 8662.776,E2 8662.776} C_VEL
LIN {X 0,Y 454.093,Z 972.763,A -85,B 0,C 180,E1 8662.042,E2 8662.042} C_VEL
LIN {X 0,Y 459.332,Z 950.82,A -85,B 0,C 180,E1 8661.393,E2 8661.393} C_VEL
LIN {X 0,Y 464.65,Z 923.43,A -85,B 0,C 180,E1 8660.755,E2 8660.755} C_VEL
LIN {X 0,Y 468.212,Z 897.253,A -85,B 0,C 180,E1 8660.287,E2 8660.287} C_VEL
LIN {X 0,Y 483.13,Z 727.489,A -85,B 0,C 180,E1 8657.686,E2 8657.686} C_VEL
LIN {X 0,Y 490.155,Z 648.201,A -85,B 0,C 180,E1 8656.472,E2 8656.472} C_VEL
LIN {X 0,Y 485.267,Z 639.895,A -85,B 0,C 180,E1 8653.889,E2 8653.889} C_VEL
LIN {X 0,Y 481.203,Z 633.094,A -85,B 0,C 180,E1 8651.264,E2 8651.264} C_VEL
LIN {X 0,Y 478.822,Z 629.2,A -85,B 0,C 180,E1 8649.374,E2 8649.374} C_VEL
LIN {X 0,Y 476.084,Z 624.626,A -85,B 0,C 180,E1 8646.512,E2 8646.512} C_VEL
LIN {X 0,Y 473.96,Z 620.952,A -85,B 0,C 180,E1 8642.539,E2 8642.539} C_VEL
LIN {X 0,Y 473.757,Z 619.601,A -85,B 0,C 180,E1 8641.088,E2 8641.088} C_VEL
LIN {X 0,Y 473.816,Z 619.824,A -85,B 0,C 180,E1 8638.549,E2 8638.549} C_VEL
LIN {X 0,Y 475.251,Z 623.77,A -85,B 0,C 180,E1 8634.688,E2 8634.688} C_VEL
LIN {X 0,Y 476.511,Z 625.342,A -85,B 0,C 180,E1 8633.07,E2 8633.07} C_VEL
LIN {X 0,Y 479.649,Z 630.552,A -85,B 0,C 180,E1 8630.036,E2 8630.036} C_VEL
LIN {X 0,Y 482.523,Z 635.399,A -85,B 0,C 180,E1 8627.919,E2 8627.919} C_VEL
LIN {X 0,Y 486.48,Z 641.838,A -85,B 0,C 180,E1 8625.539,E2 8625.539} C_VEL
LIN {X 0,Y 490.244,Z 648.438,A -85,B 0,C 180,E1 8623.589,E2 8623.589} C_VEL
LIN {X 0,Y 471.299,Z 865.047,A -85,B 0,C 180,E1 8620.293,E2 8620.293} C_VEL
LIN {X 0,Y 467.174,Z 908.723,A -85,B 0,C 180,E1 8619.602,E2 8619.602} C_VEL
LIN {X 0,Y 462.797,Z 936.048,A -85,B 0,C 180,E1 8619.076,E2 8619.076} C_VEL
LIN {X 0,Y 458.402,Z 957.5,A -85,B 0,C 180,E1 8618.561,E2 8618.561} C_VEL
LIN {X 0,Y 453.337,Z 978.24,A -85,B 0,C 180,E1 8617.95,E2 8617.95} C_VEL
LIN {X 0,Y 446.985,Z 1000.618,A -85,B 0,C 180,E1 8617.149,E2 8617.149} C_VEL
LIN {X 0,Y 437.938,Z 1027.831,A -85,B 0,C 180,E1 8615.946,E2 8615.946} C_VEL
LIN {X 0,Y 429.821,Z 1049.124,A -85,B 0,C 180,E1 8614.799,E2 8614.799} C_VEL
LIN {X 0,Y 421.912,Z 1068.029,A -85,B 0,C 180,E1 8613.6,E2 8613.6} C_VEL
LIN {X 0,Y 413.472,Z 1086.51,A -85,B 0,C 180,E1 8612.249,E2 8612.249} C_VEL
LIN {X 0,Y 402.855,Z 1108.052,A -85,B 0,C 180,E1 8610.401,E2 8610.401} C_VEL
LIN {X 0,Y 391.225,Z 1129.53,A -85,B 0,C 180,E1 8608.178,E2 8608.178} C_VEL
LIN {X 0,Y 381.625,Z 1146.2,A -85,B 0,C 180,E1 8606.145,E2 8606.145} C_VEL
LIN {X 0,Y 372.228,Z 1161.774,A -85,B 0,C 180,E1 8603.944,E2 8603.944} C_VEL
LIN {X 0,Y 362.312,Z 1177.599,A -85,B 0,C 180,E1 8601.342,E2 8601.342} C_VEL
LIN {X 0,Y 350.067,Z 1196.452,A -85,B 0,C 180,E1 8597.617,E2 8597.617} C_VEL
LIN {X 0,Y 341.217,Z 1209.797,A -85,B 0,C 180,E1 8594.446,E2 8594.446} C_VEL
LIN {X 0,Y 333.367,Z 1221.64,A -85,B 0,C 180,E1 8591.163,E2 8591.163} C_VEL
LIN {X 0,Y 325.521,Z 1233.728,A -85,B 0,C 180,E1 8587.229,E2 8587.229} C_VEL
LIN {X 0,Y 318.119,Z 1245.635,A -85,B 0,C 180,E1 8582.504,E2 8582.504} C_VEL
LIN {X 0,Y 313.208,Z 1254.188,A -85,B 0,C 180,E1 8578.395,E2 8578.395} C_VEL
LIN {X 0,Y 309.645,Z 1261.15,A -85,B 0,C 180,E1 8574.407,E2 8574.407} C_VEL
LIN {X 0,Y 306.949,Z 1267.238,A -85,B 0,C 180,E1 8570.193,E2 8570.193} C_VEL
LIN {X 0,Y 305.024,Z 1272.969,A -85,B 0,C 180,E1 8565.197,E2 8565.197} C_VEL
LIN {X 0,Y 304.159,Z 1276.781,A -85,B 0,C 180,E1 8560.411,E2 8560.411} C_VEL
LIN {X 0,Y 303.956,Z 1278.915,A -85,B 0,C 180,E1 8556.416,E2 8556.416} C_VEL
LIN {X 0,Y 303.912,Z 1280.013,A -85,B 0,C 180,E1 8552.634,E2 8552.634} C_VEL
LIN {X 0,Y 303.89,Z 1280.195,A -85,B 0,C 180,E1 8548.863,E2 8548.863} C_VEL
LIN {X 0,Y 303.923,Z 1279.459,A -85,B 0,C 180,E1 8545.088,E2 8545.088} C_VEL
LIN {X 0,Y 304.053,Z 1277.688,A -85,B 0,C 180,E1 8541.104,E2 8541.104} C_VEL
LIN {X 0,Y 304.503,Z 1275.011,A -85,B 0,C 180,E1 8537.228,E2 8537.228} C_VEL
LIN {X 0,Y 305.5,Z 1271.278,A -85,B 0,C 180,E1 8533.256,E2 8533.256} C_VEL
LIN {X 0,Y 307.265,Z 1266.434,A -85,B 0,C 180,E1 8529.22,E2 8529.22} C_VEL
LIN {X 0,Y 309.949,Z 1260.496,A -85,B 0,C 180,E1 8525.2,E2 8525.2} C_VEL
LIN {X 0,Y 314.24,Z 1252.354,A -85,B 0,C 180,E1 8520.654,E2 8520.654} C_VEL
LIN {X 0,Y 320.774,Z 1241.217,A -85,B 0,C 180,E1 8515.649,E2 8515.649} C_VEL
LIN {X 0,Y 327.177,Z 1231.065,A -85,B 0,C 180,E1 8511.874,E2 8511.874} C_VEL
LIN {X 0,Y 333.953,Z 1220.683,A -85,B 0,C 180,E1 8508.566,E2 8508.566} C_VEL
LIN {X 0,Y 342.086,Z 1208.421,A -85,B 0,C 180,E1 8505.213,E2 8505.213} C_VEL
LIN {X 0,Y 352.661,Z 1192.488,A -85,B 0,C 180,E1 8501.534,E2 8501.534} C_VEL
LIN {X 0,Y 362.863,Z 1176.604,A -85,B 0,C 180,E1 8498.499,E2 8498.499} C_VEL
LIN {X 0,Y 372.335,Z 1161.467,A -85,B 0,C 180,E1 8496.024,E2 8496.024} C_VEL
LIN {X 0,Y 381.646,Z 1146.016,A -85,B 0,C 180,E1 8493.844,E2 8493.844} C_VEL
LIN {X 0,Y 391.636,Z 1128.631,A -85,B 0,C 180,E1 8491.732,E2 8491.732} C_VEL
LIN {X 0,Y 404.34,Z 1104.82,A -85,B 0,C 180,E1 8489.317,E2 8489.317} C_VEL
LIN {X 0,Y 413.837,Z 1085.472,A -85,B 0,C 180,E1 8487.682,E2 8487.682} C_VEL
LIN {X 0,Y 421.934,Z 1067.696,A -85,B 0,C 180,E1 8486.389,E2 8486.389} C_VEL
LIN {X 0,Y 429.844,Z 1048.759,A -85,B 0,C 180,E1 8485.19,E2 8485.19} C_VEL
LIN {X 0,Y 438.336,Z 1026.412,A -85,B 0,C 180,E1 8483.992,E2 8483.992} C_VEL
LIN {X 0,Y 447.006,Z 1000.075,A -85,B 0,C 180,E1 8482.838,E2 8482.838} C_VEL
LIN {X 0,Y 453.147,Z 978.422,A -85,B 0,C 180,E1 8482.063,E2 8482.063} C_VEL
LIN {X 0,Y 458.304,Z 957.298,A -85,B 0,C 180,E1 8481.441,E2 8481.441} C_VEL
LIN {X 0,Y 462.715,Z 935.706,A -85,B 0,C 180,E1 8480.924,E2 8480.924} C_VEL
LIN {X 0,Y 467.085,Z 908.188,A -85,B 0,C 180,E1 8480.396,E2 8480.396} C_VEL
LIN {X 0,Y 471.31,Z 863.104,A -85,B 0,C 180,E1 8479.684,E2 8479.684} C_VEL
LIN {X 0,Y 490.087,Z 648.257,A -85,B 0,C 180,E1 8476.414,E2 8476.414} C_VEL
LIN {X 0,Y 485.071,Z 639.718,A -85,B 0,C 180,E1 8473.774,E2 8473.774} C_VEL
LIN {X 0,Y 480.912,Z 632.784,A -85,B 0,C 180,E1 8471.088,E2 8471.088} C_VEL
LIN {X 0,Y 478.604,Z 629.016,A -85,B 0,C 180,E1 8469.257,E2 8469.257} C_VEL
LIN {X 0,Y 475.953,Z 624.54,A -85,B 0,C 180,E1 8466.514,E2 8466.514} C_VEL
LIN {X 0,Y 473.791,Z 620.83,A -85,B 0,C 180,E1 8462.661,E2 8462.661} C_VEL
LIN {X 0,Y 473.572,Z 619.546,A -85,B 0,C 180,E1 8461.452,E2 8461.452} C_VEL
LIN {X 0,Y 473.626,Z 619.674,A -85,B 0,C 180,E1 8458.064,E2 8458.064} C_VEL
LIN {X 0,Y 475.312,Z 623.901,A -85,B 0,C 180,E1 8454.083,E2 8454.083} C_VEL
LIN {X 0,Y 476.337,Z 625.156,A -85,B 0,C 180,E1 8452.825,E2 8452.825} C_VEL
LIN {X 0,Y 479.433,Z 630.327,A -85,B 0,C 180,E1 8449.85,E2 8449.85} C_VEL
LIN {X 0,Y 482.412,Z 635.266,A -85,B 0,C 180,E1 8447.673,E2 8447.673} C_VEL
LIN {X 0,Y 485.76,Z 640.802,A -85,B 0,C 180,E1 8445.638,E2 8445.638} C_VEL
LIN {X 0,Y 490.019,Z 648.069,A -85,B 0,C 180,E1 8443.424,E2 8443.424} C_VEL
LIN {X 0,Y 471.397,Z 860.876,A -85,B 0,C 180,E1 8440.186,E2 8440.186} C_VEL
LIN {X 0,Y 467.236,Z 904.995,A -85,B 0,C 180,E1 8439.489,E2 8439.489} C_VEL
LIN {X 0,Y 462.901,Z 932.224,A -85,B 0,C 180,E1 8438.959,E2 8438.959} C_VEL
LIN {X 0,Y 458.464,Z 954.031,A -85,B 0,C 180,E1 8438.423,E2 8438.423} C_VEL
LIN {X 0,Y 453.363,Z 975.028,A -85,B 0,C 180,E1 8437.785,E2 8437.785} C_VEL
LIN {X 0,Y 446.909,Z 997.798,A -85,B 0,C 180,E1 8436.95,E2 8436.95} C_VEL
LIN {X 0,Y 437.971,Z 1024.589,A -85,B 0,C 180,E1 8435.736,E2 8435.736} C_VEL
LIN {X 0,Y 430.048,Z 1045.38,A -85,B 0,C 180,E1 8434.597,E2 8434.597} C_VEL
LIN {X 0,Y 422.215,Z 1064.066,A -85,B 0,C 180,E1 8433.398,E2 8433.398} C_VEL
LIN {X 0,Y 413.97,Z 1082.144,A -85,B 0,C 180,E1 8432.058,E2 8432.058} C_VEL
LIN {X 0,Y 404.111,Z 1102.121,A -85,B 0,C 180,E1 8430.339,E2 8430.339} C_VEL
LIN {X 0,Y 392.003,Z 1124.576,A -85,B 0,C 180,E1 8428.02,E2 8428.02} C_VEL
LIN {X 0,Y 382.288,Z 1141.369,A -85,B 0,C 180,E1 8425.963,E2 8425.963} C_VEL
LIN {X 0,Y 372.701,Z 1157.141,A -85,B 0,C 180,E1 8423.718,E2 8423.718} C_VEL
LIN {X 0,Y 362.481,Z 1173.322,A -85,B 0,C 180,E1 8421.029,E2 8421.029} C_VEL
LIN {X 0,Y 350.53,Z 1191.484,A -85,B 0,C 180,E1 8417.391,E2 8417.391} C_VEL
LIN {X 0,Y 341.96,Z 1204.238,A -85,B 0,C 180,E1 8414.338,E2 8414.338} C_VEL
LIN {X 0,Y 334.262,Z 1215.652,A -85,B 0,C 180,E1 8411.159,E2 8411.159} C_VEL
LIN {X 0,Y 326.801,Z 1226.853,A -85,B 0,C 180,E1 8407.512,E2 8407.512} C_VEL
LIN {X 0,Y 318.92,Z 1239.215,A -85,B 0,C 180,E1 8402.638,E2 8402.638} C_VEL
LIN {X 0,Y 313.689,Z 1247.982,A -85,B 0,C 180,E1 8398.387,E2 8398.387} C_VEL
LIN {X 0,Y 310.01,Z 1254.868,A -85,B 0,C 180,E1 8394.388,E2 8394.388} C_VEL
LIN {X 0,Y 307.224,Z 1260.842,A -85,B 0,C 180,E1 8390.186,E2 8390.186} C_VEL
LIN {X 0,Y 305.254,Z 1266.255,A -85,B 0,C 180,E1 8385.391,E2 8385.391} C_VEL
LIN {X 0,Y 304.244,Z 1270.192,A -85,B 0,C 180,E1 8380.419,E2 8380.419} C_VEL
LIN {X 0,Y 303.985,Z 1272.347,A -85,B 0,C 180,E1 8376.237,E2 8376.237} C_VEL
LIN {X 0,Y 303.916,Z 1273.384,A -85,B 0,C 180,E1 8372.457,E2 8372.457} C_VEL
LIN {X 0,Y 303.896,Z 1273.532,A -85,B 0,C 180,E1 8368.686,E2 8368.686} C_VEL
LIN {X 0,Y 303.944,Z 1272.79,A -85,B 0,C 180,E1 8364.91,E2 8364.91} C_VEL
LIN {X 0,Y 304.117,Z 1271.156,A -85,B 0,C 180,E1 8361.116,E2 8361.116} C_VEL
LIN {X 0,Y 304.637,Z 1268.458,A -85,B 0,C 180,E1 8357.11,E2 8357.11} C_VEL
LIN {X 0,Y 305.735,Z 1264.744,A -85,B 0,C 180,E1 8353.084,E2 8353.084} C_VEL
LIN {X 0,Y 307.497,Z 1260.234,A -85,B 0,C 180,E1 8349.248,E2 8349.248} C_VEL
LIN {X 0,Y 310.402,Z 1254.143,A -85,B 0,C 180,E1 8345.047,E2 8345.047} C_VEL
LIN {X 0,Y 315.04,Z 1245.782,A -85,B 0,C 180,E1 8340.33,E2 8340.33} C_VEL
LIN {X 0,Y 321.562,Z 1235.007,A -85,B 0,C 180,E1 8335.489,E2 8335.489} C_VEL
LIN {X 0,Y 327.991,Z 1225.089,A -85,B 0,C 180,E1 8331.776,E2 8331.776} C_VEL
LIN {X 0,Y 335.245,Z 1214.252,A -85,B 0,C 180,E1 8328.318,E2 8328.318} C_VEL
LIN {X 0,Y 344.832,Z 1200.164,A -85,B 0,C 180,E1 8324.505,E2 8324.505} C_VEL
LIN {X 0,Y 355.428,Z 1184.186,A -85,B 0,C 180,E1 8320.956,E2 8320.956} C_VEL
LIN {X 0,Y 364.584,Z 1170.113,A -85,B 0,C 180,E1 8318.303,E2 8318.303} C_VEL
LIN {X 0,Y 374.313,Z 1154.682,A -85,B 0,C 180,E1 8315.804,E2 8315.804} C_VEL
LIN {X 0,Y 383.936,Z 1138.774,A -85,B 0,C 180,E1 8313.59,E2 8313.59} C_VEL
LIN {X 0,Y 386.439,Z 1133.66,A -85,B 0,C 180,E1 8312.804,E2 8312.804} C_VEL
LIN {X 0,Y 390.696,Z 1120.386,A -85,B 0,C 180,E1 8310.447,E2 8310.447} C_VEL
LIN {X 0,Y 392.93,Z 1115.578,A -85,B 0,C 180,E1 8309.852,E2 8309.852} C_VEL
LIN {X 0,Y 402.645,Z 1097.474,A -85,B 0,C 180,E1 8308.103,E2 8308.103} C_VEL
LIN {X 0,Y 411.556,Z 1079.663,A -85,B 0,C 180,E1 8306.625,E2 8306.625} C_VEL
LIN {X 0,Y 420.179,Z 1060.999,A -85,B 0,C 180,E1 8305.289,E2 8305.289} C_VEL
LIN {X 0,Y 430.194,Z 1037.113,A -85,B 0,C 180,E1 8303.833,E2 8303.833} C_VEL
LIN {X 0,Y 438.91,Z 1013.167,A -85,B 0,C 180,E1 8302.644,E2 8302.644} C_VEL
LIN {X 0,Y 445.301,Z 993.396,A -85,B 0,C 180,E1 8301.818,E2 8301.818} C_VEL
LIN {X 0,Y 451.129,Z 972.842,A -85,B 0,C 180,E1 8301.092,E2 8301.092} C_VEL
LIN {X 0,Y 456.486,Z 950.788,A -85,B 0,C 180,E1 8300.45,E2 8300.45} C_VEL
LIN {X 0,Y 461.891,Z 923.338,A -85,B 0,C 180,E1 8299.821,E2 8299.821} C_VEL
LIN {X 0,Y 465.49,Z 897.318,A -85,B 0,C 180,E1 8299.361,E2 8299.361} C_VEL
LIN {X 0,Y 481.08,Z 723.913,A -85,B 0,C 180,E1 8296.72,E2 8296.72} C_VEL
LIN {X 0,Y 487.45,Z 653.71,A -85,B 0,C 180,E1 8295.655,E2 8295.655} C_VEL
LIN {X 0,Y 482.55,Z 645.271,A -85,B 0,C 180,E1 8292.871,E2 8292.871} C_VEL
LIN {X 0,Y 479.415,Z 640.067,A -85,B 0,C 180,E1 8290.697,E2 8290.697} C_VEL
LIN {X 0,Y 477.567,Z 636.919,A -85,B 0,C 180,E1 8289.156,E2 8289.156} C_VEL
LIN {X 0,Y 475.01,Z 632.509,A -85,B 0,C 180,E1 8286.406,E2 8286.406} C_VEL
LIN {X 0,Y 472.951,Z 628.832,A -85,B 0,C 180,E1 8282.423,E2 8282.423} C_VEL
LIN {X 0,Y 472.782,Z 627.542,A -85,B 0,C 180,E1 8281.091,E2 8281.091} C_VEL
LIN {X 0,Y 472.832,Z 627.84,A -85,B 0,C 180,E1 8278.546,E2 8278.546} C_VEL
LIN {X 0,Y 474.195,Z 631.65,A -85,B 0,C 180,E1 8274.798,E2 8274.798} C_VEL
LIN {X 0,Y 475.379,Z 633.149,A -85,B 0,C 180,E1 8273.236,E2 8273.236} C_VEL
LIN {X 0,Y 478.444,Z 638.378,A -85,B 0,C 180,E1 8270.193,E2 8270.193} C_VEL
LIN {X 0,Y 481.153,Z 643.044,A -85,B 0,C 180,E1 8268.148,E2 8268.148} C_VEL
LIN {X 0,Y 484.961,Z 649.381,A -85,B 0,C 180,E1 8265.797,E2 8265.797} C_VEL
LIN {X 0,Y 487.512,Z 654.05,A -85,B 0,C 180,E1 8264.41,E2 8264.41} C_VEL
LIN {X 0,Y 468.062,Z 871.718,A -85,B 0,C 180,E1 8261.116,E2 8261.116} C_VEL
LIN {X 0,Y 464.214,Z 910.154,A -85,B 0,C 180,E1 8260.504,E2 8260.504} C_VEL
LIN {X 0,Y 459.936,Z 936.234,A -85,B 0,C 180,E1 8260.006,E2 8260.006} C_VEL
LIN {X 0,Y 455.469,Z 957.64,A -85,B 0,C 180,E1 8259.499,E2 8259.499} C_VEL
LIN {X 0,Y 450.151,Z 978.976,A -85,B 0,C 180,E1 8258.877,E2 8258.877} C_VEL
LIN {X 0,Y 442.979,Z 1003.62,A -85,B 0,C 180,E1 8257.994,E2 8257.994} C_VEL
LIN {X 0,Y 434.303,Z 1028.755,A -85,B 0,C 180,E1 8256.875,E2 8256.875} C_VEL
LIN {X 0,Y 426.407,Z 1049.04,A -85,B 0,C 180,E1 8255.792,E2 8255.792} C_VEL
LIN {X 0,Y 418.333,Z 1067.944,A -85,B 0,C 180,E1 8254.605,E2 8254.605} C_VEL
LIN {X 0,Y 409.701,Z 1086.424,A -85,B 0,C 180,E1 8253.268,E2 8253.268} C_VEL
LIN {X 0,Y 398.584,Z 1108.46,A -85,B 0,C 180,E1 8251.39,E2 8251.39} C_VEL
LIN {X 0,Y 386.582,Z 1130,A -85,B 0,C 180,E1 8249.159,E2 8249.159} C_VEL
LIN {X 0,Y 376.619,Z 1146.811,A -85,B 0,C 180,E1 8247.105,E2 8247.105} C_VEL
LIN {X 0,Y 366.784,Z 1162.615,A -85,B 0,C 180,E1 8244.856,E2 8244.856} C_VEL
LIN {X 0,Y 354.967,Z 1180.9,A -85,B 0,C 180,E1 8241.793,E2 8241.793} C_VEL
LIN {X 0,Y 343.643,Z 1197.524,A -85,B 0,C 180,E1 8238.389,E2 8238.389} C_VEL
LIN {X 0,Y 334.81,Z 1210.346,A -85,B 0,C 180,E1 8235.288,E2 8235.288} C_VEL
LIN {X 0,Y 326.49,Z 1222.407,A -85,B 0,C 180,E1 8231.875,E2 8231.875} C_VEL
LIN {X 0,Y 317.545,Z 1235.638,A -85,B 0,C 180,E1 8227.416,E2 8227.416} C_VEL
LIN {X 0,Y 310.547,Z 1246.362,A -85,B 0,C 180,E1 8222.958,E2 8222.958} C_VEL
LIN {X 0,Y 305.674,Z 1254.454,A -85,B 0,C 180,E1 8218.947,E2 8218.947} C_VEL
LIN {X 0,Y 301.926,Z 1261.387,A -85,B 0,C 180,E1 8214.85,E2 8214.85} C_VEL
LIN {X 0,Y 298.9,Z 1267.92,A -85,B 0,C 180,E1 8210.148,E2 8210.148} C_VEL
LIN {X 0,Y 296.932,Z 1273.534,A -85,B 0,C 180,E1 8204.822,E2 8204.822} C_VEL
LIN {X 0,Y 296.168,Z 1276.808,A -85,B 0,C 180,E1 8200.498,E2 8200.498} C_VEL
LIN {X 0,Y 295.956,Z 1278.896,A -85,B 0,C 180,E1 8196.395,E2 8196.395} C_VEL
LIN {X 0,Y 295.912,Z 1279.949,A -85,B 0,C 180,E1 8192.512,E2 8192.512} C_VEL
LIN {X 0,Y 295.891,Z 1280.107,A -85,B 0,C 180,E1 8188.833,E2 8188.833} C_VEL
LIN {X 0,Y 295.924,Z 1279.371,A -85,B 0,C 180,E1 8184.955,E2 8184.955} C_VEL
LIN {X 0,Y 296.062,Z 1277.599,A -85,B 0,C 180,E1 8180.861,E2 8180.861} C_VEL
LIN {X 0,Y 296.551,Z 1274.97,A -85,B 0,C 180,E1 8176.939,E2 8176.939} C_VEL
LIN {X 0,Y 297.656,Z 1271.188,A -85,B 0,C 180,E1 8172.801,E2 8172.801} C_VEL
LIN {X 0,Y 299.569,Z 1266.303,A -85,B 0,C 180,E1 8168.629,E2 8168.629} C_VEL
LIN {X 0,Y 302.441,Z 1260.339,A -85,B 0,C 180,E1 8164.497,E2 8164.497} C_VEL
LIN {X 0,Y 306.971,Z 1252.261,A -85,B 0,C 180,E1 8159.888,E2 8159.888} C_VEL
LIN {X 0,Y 313.872,Z 1241.124,A -85,B 0,C 180,E1 8154.784,E2 8154.784} C_VEL
LIN {X 0,Y 320.604,Z 1230.972,A -85,B 0,C 180,E1 8150.946,E2 8150.946} C_VEL
LIN {X 0,Y 327.675,Z 1220.589,A -85,B 0,C 180,E1 8147.59,E2 8147.59} C_VEL
LIN {X 0,Y 336.154,Z 1208.327,A -85,B 0,C 180,E1 8144.201,E2 8144.201} C_VEL
LIN {X 0,Y 347.652,Z 1191.619,A -85,B 0,C 180,E1 8140.34,E2 8140.34} C_VEL
LIN {X 0,Y 358.264,Z 1175.66,A -85,B 0,C 180,E1 8137.302,E2 8137.302} C_VEL
LIN {X 0,Y 367.67,Z 1161.082,A -85,B 0,C 180,E1 8134.927,E2 8134.927} C_VEL
LIN {X 0,Y 377.439,Z 1145.316,A -85,B 0,C 180,E1 8132.713,E2 8132.713} C_VEL
LIN {X 0,Y 389.559,Z 1124.757,A -85,B 0,C 180,E1 8130.262,E2 8130.262} C_VEL
LIN {X 0,Y 400.989,Z 1103.497,A -85,B 0,C 180,E1 8128.176,E2 8128.176} C_VEL
LIN {X 0,Y 410.429,Z 1084.641,A -85,B 0,C 180,E1 8126.605,E2 8126.605} C_VEL
LIN {X 0,Y 419.083,Z 1065.974,A -85,B 0,C 180,E1 8125.274,E2 8125.274} C_VEL
LIN {X 0,Y 428.351,Z 1044.036,A -85,B 0,C 180,E1 8123.93,E2 8123.93} C_VEL
LIN {X 0,Y 437.759,Z 1018.726,A -85,B 0,C 180,E1 8122.661,E2 8122.661} C_VEL
LIN {X 0,Y 444.695,Z 997.405,A -85,B 0,C 180,E1 8121.776,E2 8121.776} C_VEL
LIN {X 0,Y 450.479,Z 977.178,A -85,B 0,C 180,E1 8121.074,E2 8121.074} C_VEL
LIN {X 0,Y 455.693,Z 956.005,A -85,B 0,C 180,E1 8120.466,E2 8120.466} C_VEL
LIN {X 0,Y 460.479,Z 932.619,A -85,B 0,C 180,E1 8119.924,E2 8119.924} C_VEL
LIN {X 0,Y 464.901,Z 902.921,A -85,B 0,C 180,E1 8119.382,E2 8119.382} C_VEL
LIN {X 0,Y 470.993,Z 836.348,A -85,B 0,C 180,E1 8118.353,E2 8118.353} C_VEL
LIN {X 0,Y 487.359,Z 653.747,A -85,B 0,C 180,E1 8115.591,E2 8115.591} C_VEL
LIN {X 0,Y 482.443,Z 645.237,A -85,B 0,C 180,E1 8112.813,E2 8112.813} C_VEL
LIN {X 0,Y 479.283,Z 639.989,A -85,B 0,C 180,E1 8110.64,E2 8110.64} C_VEL
LIN {X 0,Y 477.347,Z 636.731,A -85,B 0,C 180,E1 8109.039,E2 8109.039} C_VEL
LIN {X 0,Y 474.877,Z 632.422,A -85,B 0,C 180,E1 8106.407,E2 8106.407} C_VEL
LIN {X 0,Y 472.777,Z 628.71,A -85,B 0,C 180,E1 8102.546,E2 8102.546} C_VEL
LIN {X 0,Y 472.572,Z 627.482,A -85,B 0,C 180,E1 8101.334,E2 8101.334} C_VEL
LIN {X 0,Y 472.639,Z 627.721,A -85,B 0,C 180,E1 8098.06,E2 8098.06} C_VEL
LIN {X 0,Y 474.428,Z 631.978,A -85,B 0,C 180,E1 8093.951,E2 8093.951} C_VEL
LIN {X 0,Y 475.25,Z 633.081,A -85,B 0,C 180,E1 8092.93,E2 8092.93} C_VEL
LIN {X 0,Y 478.158,Z 638.017,A -85,B 0,C 180,E1 8090.066,E2 8090.066} C_VEL
LIN {X 0,Y 481.068,Z 642.964,A -85,B 0,C 180,E1 8087.882,E2 8087.882} C_VEL
LIN {X 0,Y 484.871,Z 649.316,A -85,B 0,C 180,E1 8085.551,E2 8085.551} C_VEL
LIN {X 0,Y 487.287,Z 653.72,A -85,B 0,C 180,E1 8084.242,E2 8084.242} C_VEL
LIN {X 0,Y 467.908,Z 870.521,A -85,B 0,C 180,E1 8080.963,E2 8080.963} C_VEL
LIN {X 0,Y 464.124,Z 907.564,A -85,B 0,C 180,E1 8080.371,E2 8080.371} C_VEL
LIN {X 0,Y 459.97,Z 932.903,A -85,B 0,C 180,E1 8079.879,E2 8079.879} C_VEL
LIN {X 0,Y 455.494,Z 954.455,A -85,B 0,C 180,E1 8079.354,E2 8079.354} C_VEL
LIN {X 0,Y 450.183,Z 975.864,A -85,B 0,C 180,E1 8078.711,E2 8078.711} C_VEL
LIN {X 0,Y 442.841,Z 1001.139,A -85,B 0,C 180,E1 8077.783,E2 8077.783} C_VEL
LIN {X 0,Y 434.082,Z 1026.322,A -85,B 0,C 180,E1 8076.628,E2 8076.628} C_VEL
LIN {X 0,Y 426.248,Z 1046.372,A -85,B 0,C 180,E1 8075.532,E2 8075.532} C_VEL
LIN {X 0,Y 417.861,Z 1065.859,A -85,B 0,C 180,E1 8074.282,E2 8074.282} C_VEL
LIN {X 0,Y 407.578,Z 1087.713,A -85,B 0,C 180,E1 8072.636,E2 8072.636} C_VEL
LIN {X 0,Y 395.919,Z 1109.965,A -85,B 0,C 180,E1 8070.613,E2 8070.613} C_VEL
LIN {X 0,Y 386.403,Z 1126.863,A -85,B 0,C 180,E1 8068.803,E2 8068.803} C_VEL
LIN {X 0,Y 376.894,Z 1142.789,A -85,B 0,C 180,E1 8066.83,E2 8066.83} C_VEL
LIN {X 0,Y 366.986,Z 1158.581,A -85,B 0,C 180,E1 8064.557,E2 8064.557} C_VEL
LIN {X 0,Y 355.23,Z 1176.588,A -85,B 0,C 180,E1 8061.494,E2 8061.494} C_VEL
LIN {X 0,Y 344.428,Z 1192.275,A -85,B 0,C 180,E1 8058.256,E2 8058.256} C_VEL
LIN {X 0,Y 335.573,Z 1204.963,A -85,B 0,C 180,E1 8055.171,E2 8055.171} C_VEL
LIN {X 0,Y 327.601,Z 1216.314,A -85,B 0,C 180,E1 8051.95,E2 8051.95} C_VEL
LIN {X 0,Y 319.128,Z 1228.561,A -85,B 0,C 180,E1 8047.855,E2 8047.855} C_VEL
LIN {X 0,Y 311.283,Z 1240.24,A -85,B 0,C 180,E1 8043.031,E2 8043.031} C_VEL
LIN {X 0,Y 306.361,Z 1248.12,A -85,B 0,C 180,E1 8039.102,E2 8039.102} C_VEL
LIN {X 0,Y 302.479,Z 1254.959,A -85,B 0,C 180,E1 8035.037,E2 8035.037} C_VEL
LIN {X 0,Y 299.501,Z 1260.933,A -85,B 0,C 180,E1 8030.73,E2 8030.73} C_VEL
LIN {X 0,Y 297.374,Z 1266.346,A -85,B 0,C 180,E1 8025.809,E2 8025.809} C_VEL
LIN {X 0,Y 296.288,Z 1270.281,A -85,B 0,C 180,E1 8020.702,E2 8020.702} C_VEL
LIN {X 0,Y 295.994,Z 1272.436,A -85,B 0,C 180,E1 8016.406,E2 8016.406} C_VEL
LIN {X 0,Y 295.917,Z 1273.472,A -85,B 0,C 180,E1 8012.523,E2 8012.523} C_VEL
LIN {X 0,Y 295.89,Z 1273.642,A -85,B 0,C 180,E1 8008.844,E2 8008.844} C_VEL
LIN {X 0,Y 295.943,Z 1272.945,A -85,B 0,C 180,E1 8004.966,E2 8004.966} C_VEL
LIN {X 0,Y 296.135,Z 1271.244,A -85,B 0,C 180,E1 8000.875,E2 8000.875} C_VEL
LIN {X 0,Y 296.707,Z 1268.547,A -85,B 0,C 180,E1 7996.759,E2 7996.759} C_VEL
LIN {X 0,Y 297.909,Z 1264.832,A -85,B 0,C 180,E1 7992.626,E2 7992.626} C_VEL
LIN {X 0,Y 299.916,Z 1260.073,A -85,B 0,C 180,E1 7988.493,E2 7988.493} C_VEL
LIN {X 0,Y 303.054,Z 1253.933,A -85,B 0,C 180,E1 7984.189,E2 7984.189} C_VEL
LIN {X 0,Y 308.281,Z 1245.153,A -85,B 0,C 180,E1 7979.18,E2 7979.18} C_VEL
LIN {X 0,Y 314.923,Z 1234.754,A -85,B 0,C 180,E1 7974.485,E2 7974.485} C_VEL
LIN {X 0,Y 321.786,Z 1224.709,A -85,B 0,C 180,E1 7970.69,E2 7970.69} C_VEL
LIN {X 0,Y 329.423,Z 1213.773,A -85,B 0,C 180,E1 7967.173,E2 7967.173} C_VEL
LIN {X 0,Y 339.936,Z 1198.912,A -85,B 0,C 180,E1 7963.168,E2 7963.168} C_VEL
LIN {X 0,Y 350.268,Z 1183.888,A -85,B 0,C 180,E1 7959.845,E2 7959.845} C_VEL
LIN {X 0,Y 359.375,Z 1170.352,A -85,B 0,C 180,E1 7957.286,E2 7957.286} C_VEL
LIN {X 0,Y 369.418,Z 1154.912,A -85,B 0,C 180,E1 7954.779,E2 7954.779} C_VEL
LIN {X 0,Y 381.37,Z 1135.737,A -85,B 0,C 180,E1 7952.142,E2 7952.142} C_VEL
LIN {X 0,Y 392.93,Z 1115.578,A -85,B 0,C 180,E1 7949.852,E2 7949.852} C_VEL
LIN {X 0,Y 395.47,Z 1110.077,A -85,B 0,C 180,E1 7949.16,E2 7949.16} C_VEL
LIN {X 0,Y 399.843,Z 1096.583,A -85,B 0,C 180,E1 7947.103,E2 7947.103} C_VEL
LIN {X 0,Y 402.499,Z 1090.727,A -85,B 0,C 180,E1 7946.47,E2 7946.47} C_VEL
LIN {X 0,Y 413.792,Z 1067.558,A -85,B 0,C 180,E1 7944.707,E2 7944.707} C_VEL
LIN {X 0,Y 422.719,Z 1047.332,A -85,B 0,C 180,E1 7943.415,E2 7943.415} C_VEL
LIN {X 0,Y 430.32,Z 1028.373,A -85,B 0,C 180,E1 7942.38,E2 7942.38} C_VEL
LIN {X 0,Y 437.862,Z 1007.425,A -85,B 0,C 180,E1 7941.406,E2 7941.406} C_VEL
LIN {X 0,Y 446.121,Z 981.046,A -85,B 0,C 180,E1 7940.395,E2 7940.395} C_VEL
LIN {X 0,Y 452.485,Z 956.265,A -85,B 0,C 180,E1 7939.641,E2 7939.641} C_VEL
LIN {X 0,Y 457.104,Z 934.68,A -85,B 0,C 180,E1 7939.114,E2 7939.114} C_VEL
LIN {X 0,Y 460.928,Z 912.379,A -85,B 0,C 180,E1 7938.678,E2 7938.678} C_VEL
LIN {X 0,Y 464.345,Z 883.846,A -85,B 0,C 180,E1 7938.207,E2 7938.207} C_VEL
LIN {X 0,Y 484.447,Z 663.547,A -85,B 0,C 180,E1 7934.896,E2 7934.896} C_VEL
LIN {X 0,Y 484.794,Z 659.441,A -85,B 0,C 180,E1 7934.818,E2 7934.818} C_VEL
LIN {X 0,Y 480.734,Z 652.261,A -85,B 0,C 180,E1 7932.371,E2 7932.371} C_VEL
LIN {X 0,Y 478.121,Z 647.756,A -85,B 0,C 180,E1 7930.483,E2 7930.483} C_VEL
LIN {X 0,Y 476.318,Z 644.637,A -85,B 0,C 180,E1 7928.937,E2 7928.937} C_VEL
LIN {X 0,Y 473.939,Z 640.392,A -85,B 0,C 180,E1 7926.298,E2 7926.298} C_VEL
LIN {X 0,Y 471.944,Z 636.712,A -85,B 0,C 180,E1 7922.307,E2 7922.307} C_VEL
LIN {X 0,Y 471.79,Z 635.487,A -85,B 0,C 180,E1 7920.972,E2 7920.972} C_VEL
LIN {X 0,Y 471.84,Z 635.718,A -85,B 0,C 180,E1 7918.664,E2 7918.664} C_VEL
LIN {X 0,Y 473.141,Z 639.53,A -85,B 0,C 180,E1 7914.908,E2 7914.908} C_VEL
LIN {X 0,Y 474.295,Z 641.071,A -85,B 0,C 180,E1 7913.342,E2 7913.342} C_VEL
LIN {X 0,Y 477.242,Z 646.203,A -85,B 0,C 180,E1 7910.351,E2 7910.351} C_VEL
LIN {X 0,Y 479.847,Z 650.792,A -85,B 0,C 180,E1 7908.339,E2 7908.339} C_VEL
LIN {X 0,Y 483.452,Z 656.93,A -85,B 0,C 180,E1 7906.057,E2 7906.057} C_VEL
LIN {X 0,Y 484.863,Z 659.855,A -85,B 0,C 180,E1 7905.237,E2 7905.237} C_VEL
LIN {X 0,Y 465.021,Z 877.301,A -85,B 0,C 180,E1 7901.966,E2 7901.966} C_VEL
LIN {X 0,Y 461.11,Z 913.225,A -85,B 0,C 180,E1 7901.388,E2 7901.388} C_VEL
LIN {X 0,Y 457.096,Z 936.94,A -85,B 0,C 180,E1 7900.936,E2 7900.936} C_VEL
LIN {X 0,Y 452.559,Z 958.214,A -85,B 0,C 180,E1 7900.437,E2 7900.437} C_VEL
LIN {X 0,Y 447.104,Z 979.637,A -85,B 0,C 180,E1 7899.819,E2 7899.819} C_VEL
LIN {X 0,Y 439.378,Z 1005.54,A -85,B 0,C 180,E1 7898.895,E2 7898.895} C_VEL
LIN {X 0,Y 430.784,Z 1029.678,A -85,B 0,C 180,E1 7897.82,E2 7897.82} C_VEL
LIN {X 0,Y 422.706,Z 1049.949,A -85,B 0,C 180,E1 7896.743,E2 7896.743} C_VEL
LIN {X 0,Y 414.513,Z 1068.672,A -85,B 0,C 180,E1 7895.574,E2 7895.574} C_VEL
LIN {X 0,Y 405.345,Z 1087.812,A -85,B 0,C 180,E1 7894.191,E2 7894.191} C_VEL
LIN {X 0,Y 392.92,Z 1111.545,A -85,B 0,C 180,E1 7892.138,E2 7892.138} C_VEL
LIN {X 0,Y 382.215,Z 1130.204,A -85,B 0,C 180,E1 7890.195,E2 7890.195} C_VEL
LIN {X 0,Y 371.961,Z 1147.041,A -85,B 0,C 180,E1 7888.14,E2 7888.14} C_VEL
LIN {X 0,Y 361.741,Z 1162.988,A -85,B 0,C 180,E1 7885.867,E2 7885.867} C_VEL
LIN {X 0,Y 349.842,Z 1180.811,A -85,B 0,C 180,E1 7882.872,E2 7882.872} C_VEL
LIN {X 0,Y 338.113,Z 1197.434,A -85,B 0,C 180,E1 7879.455,E2 7879.455} C_VEL
LIN {X 0,Y 328.935,Z 1210.256,A -85,B 0,C 180,E1 7876.331,E2 7876.331} C_VEL
LIN {X 0,Y 320.259,Z 1222.316,A -85,B 0,C 180,E1 7872.883,E2 7872.883} C_VEL
LIN {X 0,Y 310.906,Z 1235.548,A -85,B 0,C 180,E1 7868.358,E2 7868.358} C_VEL
LIN {X 0,Y 303.547,Z 1246.271,A -85,B 0,C 180,E1 7863.819,E2 7863.819} C_VEL
LIN {X 0,Y 298.388,Z 1254.364,A -85,B 0,C 180,E1 7859.724,E2 7859.724} C_VEL
LIN {X 0,Y 294.246,Z 1261.582,A -85,B 0,C 180,E1 7855.344,E2 7855.344} C_VEL
LIN {X 0,Y 290.853,Z 1268.6,A -85,B 0,C 180,E1 7850.1,E2 7850.1} C_VEL
LIN {X 0,Y 288.928,Z 1273.769,A -85,B 0,C 180,E1 7844.832,E2 7844.832} C_VEL
LIN {X 0,Y 288.177,Z 1276.835,A -85,B 0,C 180,E1 7840.59,E2 7840.59} C_VEL
LIN {X 0,Y 287.962,Z 1278.809,A -85,B 0,C 180,E1 7836.574,E2 7836.574} C_VEL
LIN {X 0,Y 287.912,Z 1279.861,A -85,B 0,C 180,E1 7832.582,E2 7832.582} C_VEL
LIN {X 0,Y 287.893,Z 1280.019,A -85,B 0,C 180,E1 7828.8,E2 7828.8} C_VEL
LIN {X 0,Y 287.926,Z 1279.283,A -85,B 0,C 180,E1 7824.814,E2 7824.814} C_VEL
LIN {X 0,Y 288.071,Z 1277.511,A -85,B 0,C 180,E1 7820.606,E2 7820.606} C_VEL
LIN {X 0,Y 288.614,Z 1274.88,A -85,B 0,C 180,E1 7816.573,E2 7816.573} C_VEL
LIN {X 0,Y 289.865,Z 1270.961,A -85,B 0,C 180,E1 7812.188,E2 7812.188} C_VEL
LIN {X 0,Y 291.85,Z 1266.252,A -85,B 0,C 180,E1 7808.067,E2 7808.067} C_VEL
LIN {X 0,Y 294.903,Z 1260.312,A -85,B 0,C 180,E1 7803.842,E2 7803.842} C_VEL
LIN {X 0,Y 299.524,Z 1252.526,A -85,B 0,C 180,E1 7799.281,E2 7799.281} C_VEL
LIN {X 0,Y 307.049,Z 1241.031,A -85,B 0,C 180,E1 7793.88,E2 7793.88} C_VEL
LIN {X 0,Y 314.107,Z 1230.878,A -85,B 0,C 180,E1 7789.978,E2 7789.978} C_VEL
LIN {X 0,Y 321.497,Z 1220.495,A -85,B 0,C 180,E1 7786.576,E2 7786.576} C_VEL
LIN {X 0,Y 330.336,Z 1208.233,A -85,B 0,C 180,E1 7783.153,E2 7783.153} C_VEL
LIN {X 0,Y 342.278,Z 1191.524,A -85,B 0,C 180,E1 7779.269,E2 7779.269} C_VEL
LIN {X 0,Y 353.254,Z 1175.566,A -85,B 0,C 180,E1 7776.222,E2 7776.222} C_VEL
LIN {X 0,Y 362.672,Z 1161.422,A -85,B 0,C 180,E1 7773.912,E2 7773.912} C_VEL
LIN {X 0,Y 372.623,Z 1145.828,A -85,B 0,C 180,E1 7771.716,E2 7771.716} C_VEL
LIN {X 0,Y 383.812,Z 1127.363,A -85,B 0,C 180,E1 7769.497,E2 7769.497} C_VEL
LIN {X 0,Y 396.456,Z 1104.742,A -85,B 0,C 180,E1 7767.245,E2 7767.245} C_VEL
LIN {X 0,Y 406.411,Z 1085.357,A -85,B 0,C 180,E1 7765.631,E2 7765.631} C_VEL
LIN {X 0,Y 415.184,Z 1066.899,A -85,B 0,C 180,E1 7764.319,E2 7764.319} C_VEL
LIN {X 0,Y 423.529,Z 1047.667,A -85,B 0,C 180,E1 7763.136,E2 7763.136} C_VEL
LIN {X 0,Y 433.146,Z 1023.16,A -85,B 0,C 180,E1 7761.873,E2 7761.873} C_VEL
LIN {X 0,Y 441.531,Z 998.034,A -85,B 0,C 180,E1 7760.827,E2 7760.827} C_VEL
LIN {X 0,Y 447.484,Z 977.653,A -85,B 0,C 180,E1 7760.128,E2 7760.128} C_VEL
LIN {X 0,Y 452.761,Z 956.666,A -85,B 0,C 180,E1 7759.531,E2 7759.531} C_VEL
LIN {X 0,Y 457.406,Z 934.534,A -85,B 0,C 180,E1 7759.02,E2 7759.02} C_VEL
LIN {X 0,Y 461.965,Z 905.815,A -85,B 0,C 180,E1 7758.491,E2 7758.491} C_VEL
LIN {X 0,Y 466.63,Z 857.386,A -85,B 0,C 180,E1 7757.74,E2 7757.74} C_VEL
LIN {X 0,Y 484.705,Z 659.47,A -85,B 0,C 180,E1 7754.76,E2 7754.76} C_VEL
LIN {X 0,Y 480.71,Z 652.367,A -85,B 0,C 180,E1 7752.371,E2 7752.371} C_VEL
LIN {X 0,Y 477.909,Z 647.554,A -85,B 0,C 180,E1 7750.366,E2 7750.366} C_VEL
LIN {X 0,Y 476.097,Z 644.445,A -85,B 0,C 180,E1 7748.819,E2 7748.819} C_VEL
LIN {X 0,Y 473.704,Z 640.21,A -85,B 0,C 180,E1 7746.18,E2 7746.18} C_VEL
LIN {X 0,Y 471.741,Z 636.439,A -85,B 0,C 180,E1 7742.308,E2 7742.308} C_VEL
LIN {X 0,Y 471.598,Z 635.423,A -85,B 0,C 180,E1 7741.336,E2 7741.336} C_VEL
LIN {X 0,Y 471.64,Z 635.604,A -85,B 0,C 180,E1 7738.178,E2 7738.178} C_VEL
LIN {X 0,Y 473.363,Z 639.859,A -85,B 0,C 180,E1 7734.059,E2 7734.059} C_VEL
LIN {X 0,Y 474.164,Z 641.003,A -85,B 0,C 180,E1 7733.036,E2 7733.036} C_VEL
LIN {X 0,Y 477.024,Z 645.982,A -85,B 0,C 180,E1 7730.164,E2 7730.164} C_VEL
LIN {X 0,Y 479.815,Z 650.814,A -85,B 0,C 180,E1 7728.033,E2 7728.033} C_VEL
LIN {X 0,Y 483.358,Z 656.872,A -85,B 0,C 180,E1 7725.81,E2 7725.81} C_VEL
LIN {X 0,Y 484.632,Z 659.58,A -85,B 0,C 180,E1 7725.068,E2 7725.068} C_VEL
LIN {X 0,Y 464.749,Z 877.421,A -85,B 0,C 180,E1 7721.794,E2 7721.794} C_VEL
LIN {X 0,Y 460.964,Z 911.092,A -85,B 0,C 180,E1 7721.247,E2 7721.247} C_VEL
LIN {X 0,Y 457.093,Z 933.915,A -85,B 0,C 180,E1 7720.804,E2 7720.804} C_VEL
LIN {X 0,Y 452.546,Z 955.312,A -85,B 0,C 180,E1 7720.287,E2 7720.287} C_VEL
LIN {X 0,Y 446.925,Z 977.439,A -85,B 0,C 180,E1 7719.625,E2 7719.625} C_VEL
LIN {X 0,Y 438.619,Z 1004.806,A -85,B 0,C 180,E1 7718.608,E2 7718.608} C_VEL
LIN {X 0,Y 430.542,Z 1027.419,A -85,B 0,C 180,E1 7717.568,E2 7717.568} C_VEL
LIN {X 0,Y 422.94,Z 1046.467,A -85,B 0,C 180,E1 7716.536,E2 7716.536} C_VEL
LIN {X 0,Y 414.384,Z 1065.953,A -85,B 0,C 180,E1 7715.299,E2 7715.299} C_VEL
LIN {X 0,Y 404.149,Z 1087.243,A -85,B 0,C 180,E1 7713.714,E2 7713.714} C_VEL
LIN {X 0,Y 392.046,Z 1109.876,A -85,B 0,C 180,E1 7711.681,E2 7711.681} C_VEL
LIN {X 0,Y 382.48,Z 1126.46,A -85,B 0,C 180,E1 7709.922,E2 7709.922} C_VEL
LIN {X 0,Y 372.734,Z 1142.379,A -85,B 0,C 180,E1 7707.966,E2 7707.966} C_VEL
LIN {X 0,Y 362.522,Z 1158.214,A -85,B 0,C 180,E1 7705.701,E2 7705.701} C_VEL
LIN {X 0,Y 350.644,Z 1175.889,A -85,B 0,C 180,E1 7702.715,E2 7702.715} C_VEL
LIN {X 0,Y 338.875,Z 1192.42,A -85,B 0,C 180,E1 7699.301,E2 7699.301} C_VEL
LIN {X 0,Y 329.714,Z 1205.057,A -85,B 0,C 180,E1 7696.204,E2 7696.204} C_VEL
LIN {X 0,Y 321.407,Z 1216.408,A -85,B 0,C 180,E1 7692.95,E2 7692.95} C_VEL
LIN {X 0,Y 312.615,Z 1228.572,A -85,B 0,C 180,E1 7688.826,E2 7688.826} C_VEL
LIN {X 0,Y 304.405,Z 1240.203,A -85,B 0,C 180,E1 7683.95,E2 7683.95} C_VEL
LIN {X 0,Y 299.108,Z 1248.212,A -85,B 0,C 180,E1 7679.879,E2 7679.879} C_VEL
LIN {X 0,Y 294.981,Z 1255.051,A -85,B 0,C 180,E1 7675.719,E2 7675.719} C_VEL
LIN {X 0,Y 291.805,Z 1261.024,A -85,B 0,C 180,E1 7671.303,E2 7671.303} C_VEL
LIN {X 0,Y 289.445,Z 1266.639,A -85,B 0,C 180,E1 7666.048,E2 7666.048} C_VEL
LIN {X 0,Y 288.337,Z 1270.37,A -85,B 0,C 180,E1 7661.001,E2 7661.001} C_VEL
LIN {X 0,Y 288,Z 1272.524,A -85,B 0,C 180,E1 7656.584,E2 7656.584} C_VEL
LIN {X 0,Y 287.917,Z 1273.56,A -85,B 0,C 180,E1 7652.593,E2 7652.593} C_VEL
LIN {X 0,Y 287.892,Z 1273.729,A -85,B 0,C 180,E1 7648.812,E2 7648.812} C_VEL
LIN {X 0,Y 287.947,Z 1273.033,A -85,B 0,C 180,E1 7644.826,E2 7644.826} C_VEL
LIN {X 0,Y 288.149,Z 1271.332,A -85,B 0,C 180,E1 7640.62,E2 7640.62} C_VEL
LIN {X 0,Y 288.784,Z 1268.635,A -85,B 0,C 180,E1 7636.389,E2 7636.389} C_VEL
LIN {X 0,Y 290.136,Z 1264.801,A -85,B 0,C 180,E1 7632.023,E2 7632.023} C_VEL
LIN {X 0,Y 292.242,Z 1260.162,A -85,B 0,C 180,E1 7627.899,E2 7627.899} C_VEL
LIN {X 0,Y 295.591,Z 1254.023,A -85,B 0,C 180,E1 7623.487,E2 7623.487} C_VEL
LIN {X 0,Y 301.135,Z 1245.243,A -85,B 0,C 180,E1 7618.365,E2 7618.365} C_VEL
LIN {X 0,Y 308.149,Z 1234.844,A -85,B 0,C 180,E1 7613.581,E2 7613.581} C_VEL
LIN {X 0,Y 315.001,Z 1225.268,A -85,B 0,C 180,E1 7609.891,E2 7609.891} C_VEL
LIN {X 0,Y 322.894,Z 1214.432,A -85,B 0,C 180,E1 7606.336,E2 7606.336} C_VEL
LIN {X 0,Y 333.296,Z 1200.343,A -85,B 0,C 180,E1 7602.449,E2 7602.449} C_VEL
LIN {X 0,Y 344.439,Z 1184.743,A -85,B 0,C 180,E1 7598.934,E2 7598.934} C_VEL
LIN {X 0,Y 354.389,Z 1170.441,A -85,B 0,C 180,E1 7596.214,E2 7596.214} C_VEL
LIN {X 0,Y 363.86,Z 1156.327,A -85,B 0,C 180,E1 7593.907,E2 7593.907} C_VEL
LIN {X 0,Y 374.431,Z 1139.862,A -85,B 0,C 180,E1 7591.598,E2 7591.598} C_VEL
LIN {X 0,Y 387.28,Z 1118.546,A -85,B 0,C 180,E1 7589.093,E2 7589.093} C_VEL
LIN {X 0,Y 397.953,Z 1099.234,A -85,B 0,C 180,E1 7587.21,E2 7587.21} C_VEL
LIN {X 0,Y 402.499,Z 1090.727,A -85,B 0,C 180,E1 7586.47,E2 7586.47} C_VEL
LIN {X 0,Y 405.138,Z 1084.858,A -85,B 0,C 180,E1 7585.853,E2 7585.853} C_VEL
LIN {X 0,Y 409.908,Z 1069.525,A -85,B 0,C 180,E1 7583.902,E2 7583.902} C_VEL
LIN {X 0,Y 412.057,Z 1064.18,A -85,B 0,C 180,E1 7583.441,E2 7583.441} C_VEL
LIN {X 0,Y 420.702,Z 1044.72,A -85,B 0,C 180,E1 7582.238,E2 7582.238} C_VEL
LIN {X 0,Y 430.046,Z 1021.436,A -85,B 0,C 180,E1 7581.028,E2 7581.028} C_VEL
LIN {X 0,Y 438.864,Z 995.765,A -85,B 0,C 180,E1 7579.944,E2 7579.944} C_VEL
LIN {X 0,Y 445.178,Z 974.476,A -85,B 0,C 180,E1 7579.204,E2 7579.204} C_VEL
LIN {X 0,Y 450.58,Z 953.216,A -85,B 0,C 180,E1 7578.594,E2 7578.594} C_VEL
LIN {X 0,Y 455.336,Z 930.718,A -85,B 0,C 180,E1 7578.073,E2 7578.073} C_VEL
LIN {X 0,Y 460.033,Z 900.873,A -85,B 0,C 180,E1 7577.531,E2 7577.531} C_VEL
LIN {X 0,Y 465.429,Z 845.275,A -85,B 0,C 180,E1 7576.68,E2 7576.68} C_VEL
LIN {X 0,Y 482.286,Z 665.147,A -85,B 0,C 180,E1 7573.991,E2 7573.991} C_VEL
LIN {X 0,Y 478.788,Z 658.936,A -85,B 0,C 180,E1 7571.749,E2 7571.749} C_VEL
LIN {X 0,Y 476.403,Z 654.691,A -85,B 0,C 180,E1 7569.91,E2 7569.91} C_VEL
LIN {X 0,Y 474.948,Z 652.182,A -85,B 0,C 180,E1 7568.596,E2 7568.596} C_VEL
LIN {X 0,Y 472.774,Z 648.183,A -85,B 0,C 180,E1 7566.07,E2 7566.07} C_VEL
LIN {X 0,Y 470.92,Z 644.446,A -85,B 0,C 180,E1 7562.069,E2 7562.069} C_VEL
LIN {X 0,Y 470.815,Z 643.427,A -85,B 0,C 180,E1 7560.974,E2 7560.974} C_VEL
LIN {X 0,Y 470.856,Z 643.731,A -85,B 0,C 180,E1 7558.662,E2 7558.662} C_VEL
LIN {X 0,Y 472.164,Z 647.513,A -85,B 0,C 180,E1 7554.897,E2 7554.897} C_VEL
LIN {X 0,Y 473.17,Z 648.877,A -85,B 0,C 180,E1 7553.509,E2 7553.509} C_VEL
LIN {X 0,Y 475.977,Z 653.891,A -85,B 0,C 180,E1 7550.569,E2 7550.569} C_VEL
LIN {X 0,Y 478.601,Z 658.638,A -85,B 0,C 180,E1 7548.491,E2 7548.491} C_VEL
LIN {X 0,Y 482.047,Z 664.682,A -85,B 0,C 180,E1 7546.261,E2 7546.261} C_VEL
LIN {X 0,Y 482.323,Z 665.577,A -85,B 0,C 180,E1 7546.074,E2 7546.074} C_VEL
LIN {X 0,Y 462.137,Z 882.286,A -85,B 0,C 180,E1 7542.837,E2 7542.837} C_VEL
LIN {X 0,Y 458.406,Z 914.446,A -85,B 0,C 180,E1 7542.316,E2 7542.316} C_VEL
LIN {X 0,Y 454.43,Z 937.387,A -85,B 0,C 180,E1 7541.883,E2 7541.883} C_VEL
LIN {X 0,Y 449.797,Z 958.679,A -85,B 0,C 180,E1 7541.39,E2 7541.39} C_VEL
LIN {X 0,Y 443.977,Z 981.039,A -85,B 0,C 180,E1 7540.75,E2 7540.75} C_VEL
LIN {X 0,Y 435.427,Z 1008.542,A -85,B 0,C 180,E1 7539.761,E2 7539.761} C_VEL
LIN {X 0,Y 427.33,Z 1030.74,A -85,B 0,C 180,E1 7538.774,E2 7538.774} C_VEL
LIN {X 0,Y 419.611,Z 1049.719,A -85,B 0,C 180,E1 7537.776,E2 7537.776} C_VEL
LIN {X 0,Y 411.191,Z 1068.588,A -85,B 0,C 180,E1 7536.613,E2 7536.613} C_VEL
LIN {X 0,Y 401.462,Z 1088.463,A -85,B 0,C 180,E1 7535.191,E2 7535.191} C_VEL
LIN {X 0,Y 388.443,Z 1112.625,A -85,B 0,C 180,E1 7533.101,E2 7533.101} C_VEL
LIN {X 0,Y 377.644,Z 1130.954,A -85,B 0,C 180,E1 7531.191,E2 7531.191} C_VEL
LIN {X 0,Y 367.308,Z 1147.462,A -85,B 0,C 180,E1 7529.175,E2 7529.175} C_VEL
LIN {X 0,Y 356.581,Z 1163.714,A -85,B 0,C 180,E1 7526.852,E2 7526.852} C_VEL
LIN {X 0,Y 343.065,Z 1183.123,A -85,B 0,C 180,E1 7523.517,E2 7523.517} C_VEL
LIN {X 0,Y 332.182,Z 1198.049,A -85,B 0,C 180,E1 7520.395,E2 7520.395} C_VEL
LIN {X 0,Y 322.7,Z 1210.804,A -85,B 0,C 180,E1 7517.242,E2 7517.242} C_VEL
LIN {X 0,Y 313.296,Z 1223.38,A -85,B 0,C 180,E1 7513.57,E2 7513.57} C_VEL
LIN {X 0,Y 303.286,Z 1236.845,A -85,B 0,C 180,E1 7508.776,E2 7508.776} C_VEL
LIN {X 0,Y 296.322,Z 1246.589,A -85,B 0,C 180,E1 7504.525,E2 7504.525} C_VEL
LIN {X 0,Y 290.925,Z 1254.63,A -85,B 0,C 180,E1 7500.338,E2 7500.338} C_VEL
LIN {X 0,Y 286.53,Z 1261.875,A -85,B 0,C 180,E1 7495.798,E2 7495.798} C_VEL
LIN {X 0,Y 282.801,Z 1269.153,A -85,B 0,C 180,E1 7490.05,E2 7490.05} C_VEL
LIN {X 0,Y 280.971,Z 1273.842,A -85,B 0,C 180,E1 7485.05,E2 7485.05} C_VEL
LIN {X 0,Y 280.218,Z 1276.746,A -85,B 0,C 180,E1 7480.895,E2 7480.895} C_VEL
LIN {X 0,Y 279.966,Z 1278.721,A -85,B 0,C 180,E1 7476.762,E2 7476.762} C_VEL
LIN {X 0,Y 279.913,Z 1279.751,A -85,B 0,C 180,E1 7472.861,E2 7472.861} C_VEL
LIN {X 0,Y 279.894,Z 1279.932,A -85,B 0,C 180,E1 7468.766,E2 7468.766} C_VEL
LIN {X 0,Y 279.928,Z 1279.195,A -85,B 0,C 180,E1 7464.666,E2 7464.666} C_VEL
LIN {X 0,Y 280.073,Z 1277.537,A -85,B 0,C 180,E1 7460.542,E2 7460.542} C_VEL
LIN {X 0,Y 280.687,Z 1274.79,A -85,B 0,C 180,E1 7456.186,E2 7456.186} C_VEL
LIN {X 0,Y 281.988,Z 1271.007,A -85,B 0,C 180,E1 7451.813,E2 7451.813} C_VEL
LIN {X 0,Y 284.171,Z 1266.16,A -85,B 0,C 180,E1 7447.442,E2 7447.442} C_VEL
LIN {X 0,Y 287.263,Z 1260.526,A -85,B 0,C 180,E1 7443.314,E2 7443.314} C_VEL
LIN {X 0,Y 291.869,Z 1253.146,A -85,B 0,C 180,E1 7438.844,E2 7438.844} C_VEL
LIN {X 0,Y 299.066,Z 1242.731,A -85,B 0,C 180,E1 7433.683,E2 7433.683} C_VEL
LIN {X 0,Y 307.321,Z 1231.303,A -85,B 0,C 180,E1 7429.154,E2 7429.154} C_VEL
LIN {X 0,Y 315.431,Z 1220.401,A -85,B 0,C 180,E1 7425.524,E2 7425.524} C_VEL
LIN {X 0,Y 324.152,Z 1208.778,A -85,B 0,C 180,E1 7422.238,E2 7422.238} C_VEL
LIN {X 0,Y 336.028,Z 1192.859,A -85,B 0,C 180,E1 7418.455,E2 7418.455} C_VEL
LIN {X 0,Y 347.782,Z 1176.321,A -85,B 0,C 180,E1 7415.259,E2 7415.259} C_VEL
LIN {X 0,Y 358.084,Z 1161.328,A -85,B 0,C 180,E1 7412.804,E2 7412.804} C_VEL
